  Call Extruder 0.17021
  MoveL (T15090) to (121.16, 113.18, 16.7) mm, rotated rx 180 ry 0 rz -180 deg; joints [1.945, 71.271, -37.578, 3.503, -33.743, -2.914]
  Call Extruder 0.01769
  MoveL (T15091) to (121.16, 113.76, 16.7) mm, rotated rx 180 ry 0 rz -180 deg; joints [1.945, 71.271, -37.578, 3.503, -33.743, -2.914]
  Call Extruder 0.17022
  MoveL (T15092) to (117.22, 109.83, 16.7) mm, rotated rx 180 ry 0 rz -180 deg; joints [3.284, 67.92, -31.274, 5.491, -36.773, -4.403]
  Call Extruder 0.01768
  MoveL (T15093) to (117.22, 110.41, 16.7) mm, rotated rx 180 ry 0 rz -180 deg; joints [3.284, 67.92, -31.274, 5.491, -36.773, -4.403]
  Call Extruder 0.17023
  MoveL (T15094) to (121.16, 114.34, 16.7) mm, rotated rx 180 ry 0 rz -180 deg; joints [3.287, 67.763, -30.978, 5.479, -36.911, -4.386]
  Call Extruder 0.01769
  MoveL (T15095) to (121.16, 114.92, 16.7) mm, rotated rx 180 ry 0 rz -180 deg; joints [3.287, 67.763, -30.978, 5.479, -36.911, -4.386]
  Call Extruder 0.11203
  MoveL (T15096) to (118.57, 112.33, 16.7) mm, rotated rx 180 ry 0 rz -180 deg; joints [1.884, 71.265, -37.567, 3.392, -33.745, -2.822]
  Call Extruder 0.01251
  MoveL (T15097) to (118.28, 112.62, 16.7) mm, rotated rx 180 ry 0 rz -180 deg; joints [1.823, 71.259, -37.556, 3.282, -33.747, -2.73]
  Call Extruder 0.12455
  MoveL (T15098) to (121.16, 115.5, 16.7) mm, rotated rx 180 ry 0 rz -180 deg; joints [1.823, 71.259, -37.556, 3.282, -33.747, -2.73]
  Call Extruder 0.01769
  MoveL (T15099) to (121.16, 116.08, 16.7) mm, rotated rx 180 ry 0 rz -180 deg; joints [3.291, 67.607, -30.685, 5.468, -37.048, -4.369]
  Call Extruder 0.13707
  MoveL (T15100) to (117.99, 112.91, 16.7) mm, rotated rx 180 ry 0 rz -180 deg; joints [3.295, 67.452, -30.393, 5.456, -37.184, -4.352]
  Call Extruder 0.01251
  MoveL (T15101) to (117.7, 113.2, 16.7) mm, rotated rx 180 ry 0 rz -180 deg; joints [3.295, 67.452, -30.393, 5.456, -37.184, -4.352]
  Call Extruder 0.1496
  MoveL (T15102) to (121.16, 116.65, 16.7) mm, rotated rx 180 ry 0 rz -180 deg; joints [3.295, 67.452, -30.393, 5.456, -37.184, -4.352]
  Call Extruder 0.01769
  MoveL (T15103) to (121.16, 117.23, 16.7) mm, rotated rx 180 ry 0 rz -180 deg; joints [1.762, 71.254, -37.545, 3.172, -33.75, -2.639]
  Call Extruder 0.16212
  MoveL (T15104) to (117.41, 113.48, 16.7) mm, rotated rx 180 ry 0 rz -180 deg; joints [1.762, 71.254, -37.545, 3.172, -33.75, -2.639]
  Call Extruder 0.00725
  MoveL (T15105) to (117.24, 113.65, 16.7) mm, rotated rx 180 ry 0 rz -180 deg; joints [1.701, 71.248, -37.534, 3.062, -33.752, -2.547]
  Call Extruder 0.00169
  MoveL (T15106) to (117.22, 113.7, 16.7) mm, rotated rx 180 ry 0 rz -180 deg; joints [1.701, 71.248, -37.534, 3.062, -33.752, -2.547]
  Call Extruder 0.00524
  MoveL (T15107) to (117.22, 113.88, 16.7) mm, rotated rx 180 ry 0 rz -180 deg; joints [3.298, 67.297, -30.102, 5.445, -37.32, -4.335]
  Call Extruder 0.17028
  MoveL (T15108) to (121.16, 117.81, 16.7) mm, rotated rx 180 ry 0 rz -180 deg; joints [3.298, 67.297, -30.102, 5.445, -37.32, -4.335]
  Call Extruder 0.01769
  MoveL (T15109) to (121.16, 118.39, 16.7) mm, rotated rx 180 ry 0 rz -180 deg; joints [3.302, 67.144, -29.813, 5.434, -37.455, -4.319]
  Call Extruder 0.1703
  MoveL (T15110) to (117.22, 114.45, 16.7) mm, rotated rx 180 ry 0 rz -180 deg; joints [3.302, 67.144, -29.813, 5.434, -37.455, -4.319]
  Call Extruder 0.01768
  MoveL (T15111) to (117.22, 115.03, 16.7) mm, rotated rx 180 ry 0 rz -180 deg; joints [3.302, 67.144, -29.813, 5.434, -37.455, -4.319]
  Call Extruder 0.17031
  MoveL (T15112) to (121.16, 118.97, 16.7) mm, rotated rx 180 ry 0 rz -180 deg; joints [1.64, 71.243, -37.525, 2.952, -33.754, -2.455]
  Call Extruder 0.01769
  MoveL (T15113) to (121.16, 119.55, 16.7) mm, rotated rx 180 ry 0 rz -180 deg; joints [1.64, 71.243, -37.525, 2.952, -33.754, -2.455]
  Call Extruder 0.17032
  MoveL (T15114) to (117.22, 115.61, 16.7) mm, rotated rx 180 ry 0 rz -180 deg; joints [1.64, 71.243, -37.525, 2.952, -33.754, -2.455]
  Call Extruder 0.01768
  MoveL (T15115) to (117.22, 116.19, 16.7) mm, rotated rx 180 ry 0 rz -180 deg; joints [1.579, 71.238, -37.515, 2.842, -33.756, -2.364]
  Call Extruder 0.17064
  MoveL (T15116) to (121.16, 120.14, 16.7) mm, rotated rx 180 ry 0 rz -180 deg; joints [1.579, 71.238, -37.515, 2.842, -33.756, -2.364]
  Call Extruder 0.01728
  MoveL (T15117) to (120.59, 120.14, 16.7) mm, rotated rx 180 ry 0 rz -180 deg; joints [3.305, 66.991, -29.526, 5.424, -37.589, -4.303]
  Call Extruder 0.14591
  MoveL (T15118) to (117.22, 116.76, 16.7) mm, rotated rx 180 ry 0 rz -180 deg; joints [3.305, 66.991, -29.526, 5.424, -37.589, -4.303]
  Call Extruder 0.01768
  MoveL (T15119) to (117.22, 117.34, 16.7) mm, rotated rx 180 ry 0 rz -180 deg; joints [3.309, 66.839, -29.241, 5.413, -37.722, -4.287]
  Call Extruder 0.12086
  MoveL (T15120) to (120.01, 120.14, 16.7) mm, rotated rx 180 ry 0 rz -180 deg; joints [3.309, 66.839, -29.241, 5.413, -37.722, -4.287]
  Call Extruder 0.01771
  MoveL (T15121) to (119.43, 120.14, 16.7) mm, rotated rx 180 ry 0 rz -180 deg; joints [3.309, 66.839, -29.241, 5.413, -37.722, -4.287]
  Call Extruder 0.10375
  MoveL (T15122) to (117.03, 117.74, 16.7) mm, rotated rx 180 ry 0 rz -180 deg; joints [3.309, 66.839, -29.241, 5.413, -37.722, -4.287]
  Set speed (45.0 mm/s)
  Call Extruder -1.6
  MoveL (T15123) to (117.03, 117.74, 16.7) mm, rotated rx 180 ry 0 rz -180 deg; joints [1.518, 71.233, -37.506, 2.732, -33.757, -2.272]
  Set speed (120.0 mm/s)
  MoveL (T15124) to (117.03, 117.74, 16.7) mm, rotated rx 180 ry 0 rz -180 deg; joints [1.518, 71.233, -37.506, 2.732, -33.757, -2.272]
  Call Extruder -0.38
  MoveL (T15125) to (117.79, 118.49, 16.7) mm, rotated rx 180 ry 0 rz -180 deg; joints [1.457, 71.228, -37.497, 2.622, -33.759, -2.181]
  Set speed (45.0 mm/s)
  Call Extruder -0.02
  MoveL (T15126) to (117.79, 118.49, 16.7) mm, rotated rx 180 ry 0 rz -180 deg; joints [1.457, 71.228, -37.497, 2.622, -33.759, -2.181]
  Set speed (150.0 mm/s)
  MoveL (T15127) to (117.79, 118.49, 18.7) mm, rotated rx 180 ry 0 rz -180 deg; joints [3.313, 66.688, -28.957, 5.403, -37.855, -4.271]
  MoveL (T15128) to (116.49, 107.94, 18.7) mm, rotated rx 180 ry 0 rz -180 deg; joints [3.313, 66.688, -28.957, 5.403, -37.855, -4.271]
  MoveL (T15129) to (116.49, 107.94, 16.7) mm, rotated rx 180 ry 0 rz -180 deg; joints [3.313, 66.688, -28.957, 5.403, -37.855, -4.271]
  Set speed (40.0 mm/s)
  Call Extruder 2.0
  MoveL (T15130) to (116.49, 107.94, 16.7) mm, rotated rx 180 ry 0 rz -180 deg; joints [3.313, 66.688, -28.957, 5.403, -37.855, -4.271]
  Set speed (37.7 mm/s)
  MoveL (T15131) to (116.49, 107.94, 16.7) mm, rotated rx 180 ry 0 rz -180 deg; joints [3.316, 66.538, -28.675, 5.393, -37.986, -4.255]
  Call Extruder 0.17708
  MoveL (T15132) to (112.39, 103.84, 16.7) mm, rotated rx 180 ry 0 rz -180 deg; joints [3.316, 66.538, -28.675, 5.393, -37.986, -4.255]
  Call Extruder 0.01769
  MoveL (T15133) to (111.82, 103.84, 16.7) mm, rotated rx 180 ry 0 rz -180 deg; joints [1.396, 71.223, -37.488, 2.512, -33.761, -2.089]
  Call Extruder 0.16915
  MoveL (T15134) to (115.72, 107.75, 16.7) mm, rotated rx 180 ry 0 rz -180 deg; joints [1.396, 71.223, -37.488, 2.512, -33.761, -2.089]
  Call Extruder 0.01769
  MoveL (T15135) to (115.15, 107.75, 16.7) mm, rotated rx 180 ry 0 rz -180 deg; joints [1.397, 71.043, -37.148, 2.505, -33.92, -2.079]
  Call Extruder 0.16915
  MoveL (T15136) to (111.24, 103.84, 16.7) mm, rotated rx 180 ry 0 rz -180 deg; joints [1.397, 71.043, -37.148, 2.505, -33.92, -2.079]
  Call Extruder 0.01769
  MoveL (T15137) to (110.66, 103.84, 16.7) mm, rotated rx 180 ry 0 rz -180 deg; joints [3.253, 66.53, -28.659, 5.29, -37.989, -4.174]
  Call Extruder 0.16915
  MoveL (T15138) to (114.57, 107.75, 16.7) mm, rotated rx 180 ry 0 rz -180 deg; joints [3.253, 66.53, -28.659, 5.29, -37.989, -4.174]
  Call Extruder 0.01769
  MoveL (T15139) to (113.99, 107.75, 16.7) mm, rotated rx 180 ry 0 rz -180 deg; joints [3.191, 66.521, -28.643, 5.188, -37.992, -4.093]
  Call Extruder 0.16915
  MoveL (T15140) to (110.08, 103.84, 16.7) mm, rotated rx 180 ry 0 rz -180 deg; joints [3.191, 66.521, -28.643, 5.188, -37.992, -4.093]
  Call Extruder 0.01769
  MoveL (T15141) to (109.5, 103.84, 16.7) mm, rotated rx 180 ry 0 rz -180 deg; joints [1.399, 70.864, -36.811, 2.497, -34.078, -2.069]
  Call Extruder 0.11483
  MoveL (T15142) to (112.16, 106.5, 16.7) mm, rotated rx 180 ry 0 rz -180 deg; joints [1.399, 70.864, -36.811, 2.497, -34.078, -2.069]
  Call Extruder 0.01251
  MoveL (T15143) to (111.87, 106.79, 16.7) mm, rotated rx 180 ry 0 rz -180 deg; joints [1.4, 70.686, -36.477, 2.49, -34.235, -2.059]
  Call Extruder 0.12733
  MoveL (T15144) to (108.92, 103.84, 16.7) mm, rotated rx 180 ry 0 rz -180 deg; joints [1.4, 70.686, -36.477, 2.49, -34.235, -2.059]
  Call Extruder 0.01769
  MoveL (T15145) to (108.35, 103.84, 16.7) mm, rotated rx 180 ry 0 rz -180 deg; joints [3.128, 66.513, -28.627, 5.085, -37.995, -4.011]
  Call Extruder 0.13984
  MoveL (T15146) to (111.58, 107.08, 16.7) mm, rotated rx 180 ry 0 rz -180 deg; joints [3.128, 66.513, -28.627, 5.085, -37.995, -4.011]
  Call Extruder 0.01251
  MoveL (T15147) to (111.29, 107.36, 16.7) mm, rotated rx 180 ry 0 rz -180 deg; joints [3.065, 66.505, -28.612, 4.982, -37.998, -3.93]
  Call Extruder 0.15235
  MoveL (T15148) to (107.77, 103.84, 16.7) mm, rotated rx 180 ry 0 rz -180 deg; joints [3.065, 66.505, -28.612, 4.982, -37.998, -3.93]
  Call Extruder 0.01769
  MoveL (T15149) to (107.19, 103.84, 16.7) mm, rotated rx 180 ry 0 rz -180 deg; joints [1.402, 70.51, -36.145, 2.483, -34.39, -2.049]
  Call Extruder 0.16485
  MoveL (T15150) to (111, 107.65, 16.7) mm, rotated rx 180 ry 0 rz -180 deg; joints [1.402, 70.51, -36.145, 2.483, -34.39, -2.049]
  Call Extruder 0.00339
  MoveL (T15151) to (110.92, 107.73, 16.7) mm, rotated rx 180 ry 0 rz -180 deg; joints [1.402, 70.51, -36.145, 2.483, -34.39, -2.049]
  Call Extruder 0.00168
  MoveL (T15152) to (110.87, 107.75, 16.7) mm, rotated rx 180 ry 0 rz -180 deg; joints [1.403, 70.335, -35.816, 2.476, -34.544, -2.039]
  Call Extruder 0.0107
  MoveL (T15153) to (110.52, 107.75, 16.7) mm, rotated rx 180 ry 0 rz -180 deg; joints [1.403, 70.335, -35.816, 2.476, -34.544, -2.039]
  Call Extruder 0.16915
  MoveL (T15154) to (106.61, 103.84, 16.7) mm, rotated rx 180 ry 0 rz -180 deg; joints [1.403, 70.335, -35.816, 2.476, -34.544, -2.039]
  Call Extruder 0.01769
  MoveL (T15155) to (106.03, 103.84, 16.7) mm, rotated rx 180 ry 0 rz -180 deg; joints [3.002, 66.497, -28.597, 4.88, -38, -3.849]
  Call Extruder 0.16915
  MoveL (T15156) to (109.94, 107.75, 16.7) mm, rotated rx 180 ry 0 rz -180 deg; joints [3.002, 66.497, -28.597, 4.88, -38, -3.849]
  Call Extruder 0.01769
  MoveL (T15157) to (109.36, 107.75, 16.7) mm, rotated rx 180 ry 0 rz -180 deg; joints [3.002, 66.497, -28.597, 4.88, -38, -3.849]
  Call Extruder 0.16915
  MoveL (T15158) to (105.45, 103.84, 16.7) mm, rotated rx 180 ry 0 rz -180 deg; joints [3.002, 66.497, -28.597, 4.88, -38, -3.849]
  Call Extruder 0.01769
  MoveL (T15159) to (104.88, 103.84, 16.7) mm, rotated rx 180 ry 0 rz -180 deg; joints [2.939, 66.489, -28.583, 4.777, -38.003, -3.768]
  Call Extruder 0.16915
  MoveL (T15160) to (108.79, 107.75, 16.7) mm, rotated rx 180 ry 0 rz -180 deg; joints [2.939, 66.489, -28.583, 4.777, -38.003, -3.768]
  Call Extruder 0.01769
  MoveL (T15161) to (108.21, 107.75, 16.7) mm, rotated rx 180 ry 0 rz -180 deg; joints [2.939, 66.489, -28.583, 4.777, -38.003, -3.768]
  Call Extruder 0.16005
  MoveL (T15162) to (104.51, 104.06, 16.7) mm, rotated rx 180 ry 0 rz -180 deg; joints [1.405, 70.161, -35.489, 2.469, -34.697, -2.03]
  Call Extruder 0.01768
  MoveL (T15163) to (104.51, 104.63, 16.7) mm, rotated rx 180 ry 0 rz -180 deg; joints [1.405, 70.161, -35.489, 2.469, -34.697, -2.03]
  Call Extruder 0.13504
  MoveL (T15164) to (107.63, 107.75, 16.7) mm, rotated rx 180 ry 0 rz -180 deg; joints [1.406, 69.989, -35.164, 2.462, -34.849, -2.021]
  Call Extruder 0.01769
  MoveL (T15165) to (107.05, 107.75, 16.7) mm, rotated rx 180 ry 0 rz -180 deg; joints [1.406, 69.989, -35.164, 2.462, -34.849, -2.021]
  Call Extruder 0.11004
  MoveL (T15166) to (104.51, 105.21, 16.7) mm, rotated rx 180 ry 0 rz -180 deg; joints [2.876, 66.482, -28.569, 4.675, -38.006, -3.686]
  Call Extruder 0.01678
  MoveL (T15167) to (104.51, 105.76, 16.7) mm, rotated rx 180 ry 0 rz -180 deg; joints [2.876, 66.482, -28.569, 4.675, -38.006, -3.686]
  Call Extruder 0.00167
  MoveL (T15168) to (104.53, 105.81, 16.7) mm, rotated rx 180 ry 0 rz -180 deg; joints [2.876, 66.482, -28.569, 4.675, -38.006, -3.686]
  Call Extruder 0.09205
  MoveL (T15169) to (106.66, 107.94, 16.7) mm, rotated rx 180 ry 0 rz -180 deg; joints [2.813, 66.474, -28.555, 4.572, -38.008, -3.605]
  Set speed (45.0 mm/s)
  Call Extruder -1.6
  MoveL (T15170) to (106.66, 107.94, 16.7) mm, rotated rx 180 ry 0 rz -180 deg; joints [2.813, 66.474, -28.555, 4.572, -38.008, -3.605]
  Set speed (120.0 mm/s)
  MoveL (T15171) to (106.66, 107.94, 16.7) mm, rotated rx 180 ry 0 rz -180 deg; joints [1.408, 69.817, -34.842, 2.455, -35, -2.012]
  Call Extruder -0.38
  MoveL (T15172) to (105.9, 107.18, 16.7) mm, rotated rx 180 ry 0 rz -180 deg; joints [1.408, 69.817, -34.842, 2.455, -35, -2.012]
  Set speed (45.0 mm/s)
  Call Extruder -0.02
  MoveL (T15173) to (105.9, 107.18, 16.7) mm, rotated rx 180 ry 0 rz -180 deg; joints [1.408, 69.817, -34.842, 2.455, -35, -2.012]
  Set speed (150.0 mm/s)
  MoveL (T15174) to (105.9, 107.18, 18.7) mm, rotated rx 180 ry 0 rz -180 deg; joints [1.409, 69.647, -34.523, 2.449, -35.149, -2.003]
  MoveL (T15175) to (104.34, 103.54, 18.7) mm, rotated rx 180 ry 0 rz -180 deg; joints [1.409, 69.647, -34.523, 2.449, -35.149, -2.003]
  MoveL (T15176) to (104.34, 103.54, 16.9) mm, rotated rx 180 ry 0 rz -180 deg; joints [2.751, 66.467, -28.541, 4.47, -38.011, -3.524]
  Set speed (40.0 mm/s)
  Call Extruder 2.0
  MoveL (T15177) to (104.34, 103.54, 16.9) mm, rotated rx 180 ry 0 rz -180 deg; joints [2.751, 66.467, -28.541, 4.47, -38.011, -3.524]
  Call Extruder 0.52159
  MoveL (T15178) to (121.46, 103.54, 16.9) mm, rotated rx 180 ry 0 rz -180 deg; joints [2.751, 66.467, -28.541, 4.47, -38.011, -3.524]
  Call Extruder 0.54596
  MoveL (T15179) to (121.46, 121.46, 16.9) mm, rotated rx 180 ry 0 rz -180 deg; joints [2.751, 66.467, -28.541, 4.47, -38.011, -3.524]
  Call Extruder 0.54596
  MoveL (T15180) to (103.54, 121.46, 16.9) mm, rotated rx 180 ry 0 rz -180 deg; joints [2.688, 66.46, -28.528, 4.367, -38.013, -3.443]
  Call Extruder 0.54596
  MoveL (T15181) to (103.54, 103.54, 16.9) mm, rotated rx 180 ry 0 rz -180 deg; joints [2.688, 66.46, -28.528, 4.367, -38.013, -3.443]
  Call Extruder 0.02254
  MoveL (T15182) to (104.28, 103.54, 16.9) mm, rotated rx 180 ry 0 rz -180 deg; joints [1.411, 69.479, -34.205, 2.442, -35.298, -1.994]
  Set speed (150.0 mm/s)
  MoveL (T15183) to (103.53, 103.13, 16.9) mm, rotated rx 180 ry 0 rz -180 deg; joints [1.411, 69.479, -34.205, 2.442, -35.298, -1.994]
  Set speed (40.0 mm/s)
  MoveL (T15184) to (103.53, 103.13, 16.9) mm, rotated rx 180 ry 0 rz -180 deg; joints [1.412, 69.311, -33.89, 2.436, -35.445, -1.985]
  Call Extruder 0.55858
  MoveL (T15185) to (121.87, 103.13, 16.9) mm, rotated rx 180 ry 0 rz -180 deg; joints [1.412, 69.311, -33.89, 2.436, -35.445, -1.985]
  Call Extruder 0.57077
  MoveL (T15186) to (121.87, 121.87, 16.9) mm, rotated rx 180 ry 0 rz -180 deg; joints [1.412, 69.311, -33.89, 2.436, -35.445, -1.985]
  Call Extruder 0.57077
  MoveL (T15187) to (103.13, 121.87, 16.9) mm, rotated rx 180 ry 0 rz -180 deg; joints [1.412, 69.311, -33.89, 2.436, -35.445, -1.985]
  Call Extruder 0.57077
  MoveL (T15188) to (103.13, 103.13, 16.9) mm, rotated rx 180 ry 0 rz -180 deg; joints [2.625, 66.453, -28.515, 4.264, -38.015, -3.362]
  Call Extruder 0.01036
  MoveL (T15189) to (103.47, 103.13, 16.9) mm, rotated rx 180 ry 0 rz -180 deg; joints [2.625, 66.453, -28.515, 4.264, -38.015, -3.362]
  Set speed (150.0 mm/s)
  MoveL (T15190) to (102.72, 102.81, 16.9) mm, rotated rx 180 ry 0 rz -180 deg; joints [2.562, 66.446, -28.502, 4.162, -38.018, -3.281]
  Set speed (25.0 mm/s)
  MoveL (T15191) to (102.72, 102.81, 16.9) mm, rotated rx 180 ry 0 rz -180 deg; joints [2.562, 66.446, -28.502, 4.162, -38.018, -3.281]
  Call Extruder 0.00259
  MoveL (T15192) to (102.72, 102.72, 16.9) mm, rotated rx 180 ry 0 rz -180 deg; joints [1.414, 69.145, -33.577, 2.43, -35.592, -1.976]
  Call Extruder 0.59557
  MoveL (T15193) to (122.28, 102.72, 16.9) mm, rotated rx 180 ry 0 rz -180 deg; joints [1.414, 69.145, -33.577, 2.43, -35.592, -1.976]
  Call Extruder 0.59557
  MoveL (T15194) to (122.28, 122.28, 16.9) mm, rotated rx 180 ry 0 rz -180 deg; joints [1.416, 68.98, -33.267, 2.424, -35.737, -1.968]
  Call Extruder 0.59557
  MoveL (T15195) to (102.72, 122.28, 16.9) mm, rotated rx 180 ry 0 rz -180 deg; joints [1.416, 68.98, -33.267, 2.424, -35.737, -1.968]
  Call Extruder 0.59115
  MoveL (T15196) to (102.72, 102.87, 16.9) mm, rotated rx 180 ry 0 rz -180 deg; joints [1.416, 68.98, -33.267, 2.424, -35.737, -1.968]
  Set speed (150.0 mm/s)
  MoveL (T15197) to (102.78, 102.75, 16.9) mm, rotated rx 180 ry 0 rz -180 deg; joints [2.499, 66.439, -28.489, 4.059, -38.02, -3.2]
  Set speed (45.0 mm/s)
  Call Extruder -1.6
  MoveL (T15198) to (102.78, 102.75, 16.9) mm, rotated rx 180 ry 0 rz -180 deg; joints [2.499, 66.439, -28.489, 4.059, -38.02, -3.2]
  Set speed (120.0 mm/s)
  MoveL (T15199) to (102.78, 102.75, 16.9) mm, rotated rx 180 ry 0 rz -180 deg; joints [2.436, 66.433, -28.477, 3.957, -38.022, -3.119]
  Call Extruder -0.05166
  MoveL (T15200) to (102.72, 102.72, 16.9) mm, rotated rx 180 ry 0 rz -180 deg; joints [2.436, 66.433, -28.477, 3.957, -38.022, -3.119]
  Call Extruder -0.32834
  MoveL (T15201) to (103.65, 102.72, 16.9) mm, rotated rx 180 ry 0 rz -180 deg; joints [1.417, 68.816, -32.958, 2.418, -35.882, -1.96]
  Set speed (45.0 mm/s)
  Call Extruder -0.02
  MoveL (T15202) to (103.65, 102.72, 16.9) mm, rotated rx 180 ry 0 rz -180 deg; joints [1.419, 68.653, -32.652, 2.412, -36.025, -1.952]
  Set speed (150.0 mm/s)
  MoveL (T15203) to (103.65, 102.72, 18.9) mm, rotated rx 180 ry 0 rz -180 deg; joints [1.419, 68.653, -32.652, 2.412, -36.025, -1.952]
  MoveL (T15204) to (103.84, 106.29, 18.9) mm, rotated rx 180 ry 0 rz -180 deg; joints [2.373, 66.427, -28.466, 3.855, -38.024, -3.038]
  MoveL (T15205) to (103.84, 106.29, 16.9) mm, rotated rx 180 ry 0 rz -180 deg; joints [2.373, 66.427, -28.466, 3.855, -38.024, -3.038]
  Set speed (40.0 mm/s)
  Call Extruder 2.0
  MoveL (T15206) to (103.84, 106.29, 16.9) mm, rotated rx 180 ry 0 rz -180 deg; joints [2.373, 66.427, -28.466, 3.855, -38.024, -3.038]
  Set speed (50.0 mm/s)
  MoveL (T15207) to (103.84, 106.29, 16.9) mm, rotated rx 180 ry 0 rz -180 deg; joints [2.31, 66.421, -28.454, 3.752, -38.026, -2.957]
  Call Extruder 0.07441
  MoveL (T15208) to (103.84, 103.84, 16.9) mm, rotated rx 180 ry 0 rz -180 deg; joints [2.31, 66.421, -28.454, 3.752, -38.026, -2.957]
  Call Extruder 0.0111
  MoveL (T15209) to (104.1, 104.1, 16.9) mm, rotated rx 180 ry 0 rz -180 deg; joints [2.31, 66.421, -28.454, 3.752, -38.026, -2.957]
  Call Extruder 0.05294
  MoveL (T15210) to (104.1, 105.84, 16.9) mm, rotated rx 180 ry 0 rz -180 deg; joints [1.42, 68.491, -32.347, 2.407, -36.168, -1.943]
  Call Extruder 0.00661
  MoveL (T15211) to (104.18, 106.04, 16.9) mm, rotated rx 180 ry 0 rz -180 deg; joints [1.42, 68.491, -32.347, 2.407, -36.168, -1.943]
  Call Extruder 0.02065
  MoveL (T15212) to (104.66, 106.52, 16.9) mm, rotated rx 180 ry 0 rz -180 deg; joints [1.42, 68.491, -32.347, 2.407, -36.168, -1.943]
  Call Extruder 0.03528
  MoveL (T15213) to (103.84, 107.34, 16.9) mm, rotated rx 180 ry 0 rz -180 deg; joints [1.422, 68.33, -32.044, 2.401, -36.31, -1.935]
  Call Extruder 0.03385
  MoveL (T15214) to (103.84, 108.45, 16.9) mm, rotated rx 180 ry 0 rz -180 deg; joints [1.422, 68.33, -32.044, 2.401, -36.31, -1.935]
  Call Extruder 0.13495
  MoveL (T15215) to (106.98, 111.58, 16.9) mm, rotated rx 180 ry 0 rz -180 deg; joints [1.422, 68.33, -32.044, 2.401, -36.31, -1.935]
  Call Extruder 0.04156
  MoveL (T15216) to (107.6, 112.8, 16.9) mm, rotated rx 180 ry 0 rz -180 deg; joints [1.422, 68.33, -32.044, 2.401, -36.31, -1.935]
  Call Extruder 0.16166
  MoveL (T15217) to (103.84, 116.55, 16.9) mm, rotated rx 180 ry 0 rz -180 deg; joints [2.247, 66.415, -28.443, 3.65, -38.028, -2.876]
  Call Extruder 0.03385
  MoveL (T15218) to (103.84, 117.66, 16.9) mm, rotated rx 180 ry 0 rz -180 deg; joints [2.247, 66.415, -28.443, 3.65, -38.028, -2.876]
  Call Extruder 0.05612
  MoveL (T15219) to (105.15, 118.96, 16.9) mm, rotated rx 180 ry 0 rz -180 deg; joints [2.185, 66.409, -28.432, 3.547, -38.03, -2.796]
  Call Extruder 0.02709
  MoveL (T15220) to (105.15, 119.85, 16.9) mm, rotated rx 180 ry 0 rz -180 deg; joints [2.185, 66.409, -28.432, 3.547, -38.03, -2.796]
  Call Extruder 0.05612
  MoveL (T15221) to (103.84, 121.16, 16.9) mm, rotated rx 180 ry 0 rz -180 deg; joints [2.185, 66.409, -28.432, 3.547, -38.03, -2.796]
  Call Extruder 0.06345
  MoveL (T15222) to (105.93, 121.16, 16.9) mm, rotated rx 180 ry 0 rz -180 deg; joints [1.423, 68.17, -31.744, 2.396, -36.45, -1.928]
  Call Extruder 0.01096
  MoveL (T15223) to (105.67, 120.9, 16.9) mm, rotated rx 180 ry 0 rz -180 deg; joints [1.423, 68.17, -31.744, 2.396, -36.45, -1.928]
  Set speed (45.0 mm/s)
  Call Extruder -1.6
  MoveL (T15224) to (105.67, 120.9, 16.9) mm, rotated rx 180 ry 0 rz -180 deg; joints [1.425, 68.011, -31.445, 2.391, -36.59, -1.92]
  Set speed (120.0 mm/s)
  MoveL (T15225) to (105.67, 120.9, 16.9) mm, rotated rx 180 ry 0 rz -180 deg; joints [1.425, 68.011, -31.445, 2.391, -36.59, -1.92]
  Call Extruder -0.12811
  MoveL (T15226) to (105.93, 121.16, 16.9) mm, rotated rx 180 ry 0 rz -180 deg; joints [2.122, 66.403, -28.422, 3.445, -38.032, -2.715]
  Call Extruder -0.25189
  MoveL (T15227) to (105.22, 121.16, 16.9) mm, rotated rx 180 ry 0 rz -180 deg; joints [2.122, 66.403, -28.422, 3.445, -38.032, -2.715]
  Set speed (45.0 mm/s)
  Call Extruder -0.02
  MoveL (T15228) to (105.22, 121.16, 16.9) mm, rotated rx 180 ry 0 rz -180 deg; joints [2.122, 66.403, -28.422, 3.445, -38.032, -2.715]
  Set speed (150.0 mm/s)
  MoveL (T15229) to (105.22, 121.16, 18.9) mm, rotated rx 180 ry 0 rz -180 deg; joints [2.059, 66.398, -28.411, 3.342, -38.034, -2.634]
  MoveL (T15230) to (105.15, 117.23, 18.9) mm, rotated rx 180 ry 0 rz -180 deg; joints [2.059, 66.398, -28.411, 3.342, -38.034, -2.634]
  MoveL (T15231) to (105.15, 117.23, 16.9) mm, rotated rx 180 ry 0 rz -180 deg; joints [2.059, 66.398, -28.411, 3.342, -38.034, -2.634]
  Set speed (40.0 mm/s)
  Call Extruder 2.0
  MoveL (T15232) to (105.15, 117.23, 16.9) mm, rotated rx 180 ry 0 rz -180 deg; joints [1.426, 67.853, -31.148, 2.385, -36.729, -1.912]
  Set speed (50.0 mm/s)
  MoveL (T15233) to (105.15, 117.23, 16.9) mm, rotated rx 180 ry 0 rz -180 deg; joints [1.426, 67.853, -31.148, 2.385, -36.729, -1.912]
  Call Extruder 0.04143
  MoveL (T15234) to (105.15, 115.87, 16.9) mm, rotated rx 180 ry 0 rz -180 deg; joints [1.426, 67.853, -31.148, 2.385, -36.729, -1.912]
  Call Extruder 0.00661
  MoveL (T15235) to (105.23, 115.67, 16.9) mm, rotated rx 180 ry 0 rz -180 deg; joints [1.428, 67.696, -30.852, 2.38, -36.867, -1.905]
  Call Extruder 0.02637
  MoveL (T15236) to (105.84, 115.05, 16.9) mm, rotated rx 180 ry 0 rz -180 deg; joints [1.428, 67.696, -30.852, 2.38, -36.867, -1.905]
  Call Extruder 0.08606
  MoveL (T15237) to (103.84, 113.06, 16.9) mm, rotated rx 180 ry 0 rz -180 deg; joints [1.428, 67.696, -30.852, 2.38, -36.867, -1.905]
  Call Extruder 0.03385
  MoveL (T15238) to (103.84, 111.94, 16.9) mm, rotated rx 180 ry 0 rz -180 deg; joints [1.428, 67.696, -30.852, 2.38, -36.867, -1.905]
  Call Extruder 0.09463
  MoveL (T15239) to (106.04, 109.75, 16.9) mm, rotated rx 180 ry 0 rz -180 deg; joints [1.996, 66.393, -28.401, 3.24, -38.036, -2.553]
  Call Extruder 0.05062
  MoveL (T15240) to (105.29, 108.27, 16.9) mm, rotated rx 180 ry 0 rz -180 deg; joints [1.996, 66.393, -28.401, 3.24, -38.036, -2.553]
  Call Extruder 0.02377
  MoveL (T15241) to (105.1, 107.51, 16.9) mm, rotated rx 180 ry 0 rz -180 deg; joints [1.996, 66.393, -28.401, 3.24, -38.036, -2.553]
  Set speed (45.0 mm/s)
  Call Extruder -1.6
  MoveL (T15242) to (105.1, 107.51, 16.9) mm, rotated rx 180 ry 0 rz -180 deg; joints [1.933, 66.388, -28.392, 3.138, -38.037, -2.472]
  Set speed (120.0 mm/s)
  MoveL (T15243) to (105.1, 107.51, 16.9) mm, rotated rx 180 ry 0 rz -180 deg; joints [1.933, 66.388, -28.392, 3.138, -38.037, -2.472]
  Call Extruder -0.27797
  MoveL (T15244) to (105.29, 108.27, 16.9) mm, rotated rx 180 ry 0 rz -180 deg; joints [1.429, 67.54, -30.559, 2.375, -37.005, -1.897]
  Call Extruder -0.10203
  MoveL (T15245) to (105.42, 108.52, 16.9) mm, rotated rx 180 ry 0 rz -180 deg; joints [1.429, 67.54, -30.559, 2.375, -37.005, -1.897]
  Set speed (45.0 mm/s)
  Call Extruder -0.02
  MoveL (T15246) to (105.42, 108.52, 16.9) mm, rotated rx 180 ry 0 rz -180 deg; joints [1.429, 67.54, -30.559, 2.375, -37.005, -1.897]
  Set speed (150.0 mm/s)
  MoveL (T15247) to (105.42, 108.52, 18.9) mm, rotated rx 180 ry 0 rz -180 deg; joints [1.429, 67.54, -30.559, 2.375, -37.005, -1.897]
  MoveL (T15248) to (117.45, 112.15, 18.9) mm, rotated rx 180 ry 0 rz -180 deg; joints [1.431, 67.385, -30.267, 2.37, -37.141, -1.89]
  MoveL (T15249) to (117.45, 112.15, 16.9) mm, rotated rx 180 ry 0 rz -180 deg; joints [1.431, 67.385, -30.267, 2.37, -37.141, -1.89]
  Set speed (40.0 mm/s)
  Call Extruder 2.0
  MoveL (T15250) to (117.45, 112.15, 16.9) mm, rotated rx 180 ry 0 rz -180 deg; joints [1.87, 66.383, -28.382, 3.035, -38.039, -2.391]
  Set speed (50.0 mm/s)
  MoveL (T15251) to (117.45, 112.15, 16.9) mm, rotated rx 180 ry 0 rz -180 deg; joints [1.807, 66.378, -28.373, 2.933, -38.041, -2.311]
  Call Extruder 0.01607
  MoveL (T15252) to (117.83, 111.78, 16.9) mm, rotated rx 180 ry 0 rz -180 deg; joints [1.807, 66.378, -28.373, 2.933, -38.041, -2.311]
  Set speed (45.0 mm/s)
  Call Extruder -1.6
  MoveL (T15253) to (117.83, 111.78, 16.9) mm, rotated rx 180 ry 0 rz -180 deg; joints [1.807, 66.378, -28.373, 2.933, -38.041, -2.311]
  Set speed (120.0 mm/s)
  MoveL (T15254) to (117.83, 111.78, 16.9) mm, rotated rx 180 ry 0 rz -180 deg; joints [1.807, 66.378, -28.373, 2.933, -38.041, -2.311]
  Call Extruder -0.18789
  MoveL (T15255) to (117.45, 112.15, 16.9) mm, rotated rx 180 ry 0 rz -180 deg; joints [1.433, 67.231, -29.977, 2.366, -37.277, -1.883]
  Set speed (45.0 mm/s)
  Call Extruder -0.21211
  MoveL (T15256) to (117.45, 112.15, 16.9) mm, rotated rx 180 ry 0 rz -180 deg; joints [1.433, 67.231, -29.977, 2.366, -37.277, -1.883]
  Set speed (150.0 mm/s)
  MoveL (T15257) to (117.45, 112.15, 18.9) mm, rotated rx 180 ry 0 rz -180 deg; joints [1.434, 67.077, -29.689, 2.361, -37.412, -1.876]
  MoveL (T15258) to (121.34, 119.42, 18.9) mm, rotated rx 180 ry 0 rz -180 deg; joints [1.434, 67.077, -29.689, 2.361, -37.412, -1.876]
  MoveL (T15259) to (121.34, 119.42, 16.9) mm, rotated rx 180 ry 0 rz -180 deg; joints [1.744, 66.373, -28.365, 2.831, -38.042, -2.23]
  Set speed (40.0 mm/s)
  Call Extruder 2.0
  MoveL (T15260) to (121.34, 119.42, 16.9) mm, rotated rx 180 ry 0 rz -180 deg; joints [1.744, 66.373, -28.365, 2.831, -38.042, -2.23]
  Call Extruder 0.03108
  MoveL (T15261) to (120.62, 120.14, 16.9) mm, rotated rx 180 ry 0 rz -180 deg; joints [1.744, 66.373, -28.365, 2.831, -38.042, -2.23]
  Call Extruder 0.01774
  MoveL (T15262) to (120.04, 120.14, 16.9) mm, rotated rx 180 ry 0 rz -180 deg; joints [1.681, 66.369, -28.356, 2.728, -38.044, -2.149]
  Call Extruder 0.04823
  MoveL (T15263) to (121.16, 119.02, 16.9) mm, rotated rx 180 ry 0 rz -180 deg; joints [1.681, 66.369, -28.356, 2.728, -38.044, -2.149]
  Call Extruder 0.01777
  MoveL (T15264) to (121.16, 118.44, 16.9) mm, rotated rx 180 ry 0 rz -180 deg; joints [1.436, 66.925, -29.402, 2.356, -37.546, -1.869]
  Call Extruder 0.07952
  MoveL (T15265) to (119.32, 120.28, 16.9) mm, rotated rx 180 ry 0 rz -180 deg; joints [1.436, 66.925, -29.402, 2.356, -37.546, -1.869]
  Call Extruder 0.01256
  MoveL (T15266) to (119.03, 119.99, 16.9) mm, rotated rx 180 ry 0 rz -180 deg; joints [1.437, 66.773, -29.117, 2.352, -37.679, -1.862]
  Call Extruder 0.09207
  MoveL (T15267) to (121.16, 117.86, 16.9) mm, rotated rx 180 ry 0 rz -180 deg; joints [1.437, 66.773, -29.117, 2.352, -37.679, -1.862]
  Call Extruder 0.01777
  MoveL (T15268) to (121.16, 117.28, 16.9) mm, rotated rx 180 ry 0 rz -180 deg; joints [1.437, 66.773, -29.117, 2.352, -37.679, -1.862]
  Call Extruder 0.10462
  MoveL (T15269) to (118.74, 119.7, 16.9) mm, rotated rx 180 ry 0 rz -180 deg; joints [1.437, 66.773, -29.117, 2.352, -37.679, -1.862]
  Call Extruder 0.01256
  MoveL (T15270) to (118.45, 119.41, 16.9) mm, rotated rx 180 ry 0 rz -180 deg; joints [1.618, 66.364, -28.348, 2.626, -38.045, -2.069]
  Call Extruder 0.11718
  MoveL (T15271) to (121.16, 116.7, 16.9) mm, rotated rx 180 ry 0 rz -180 deg; joints [1.555, 66.36, -28.341, 2.524, -38.047, -1.988]
  Call Extruder 0.01777
  MoveL (T15272) to (121.16, 116.13, 16.9) mm, rotated rx 180 ry 0 rz -180 deg; joints [1.555, 66.36, -28.341, 2.524, -38.047, -1.988]
  Call Extruder 0.12973
  MoveL (T15273) to (118.16, 119.12, 16.9) mm, rotated rx 180 ry 0 rz -180 deg; joints [1.555, 66.36, -28.341, 2.524, -38.047, -1.988]
  Call Extruder 0.01256
  MoveL (T15274) to (117.87, 118.83, 16.9) mm, rotated rx 180 ry 0 rz -180 deg; joints [1.439, 66.623, -28.834, 2.347, -37.812, -1.855]
  Call Extruder 0.14228
  MoveL (T15275) to (121.16, 115.55, 16.9) mm, rotated rx 180 ry 0 rz -180 deg; joints [1.439, 66.623, -28.834, 2.347, -37.812, -1.855]
  Call Extruder 0.01777
  MoveL (T15276) to (121.16, 114.97, 16.9) mm, rotated rx 180 ry 0 rz -180 deg; joints [1.44, 66.473, -28.552, 2.343, -37.944, -1.848]
  Call Extruder 0.15483
  MoveL (T15277) to (117.58, 118.54, 16.9) mm, rotated rx 180 ry 0 rz -180 deg; joints [1.44, 66.473, -28.552, 2.343, -37.944, -1.848]
  Call Extruder 0.01256
  MoveL (T15278) to (117.3, 118.25, 16.9) mm, rotated rx 180 ry 0 rz -180 deg; joints [1.512, 66.311, -28.247, 2.452, -38.089, -1.931]
  Call Extruder 0.16739
  MoveL (T15279) to (121.16, 114.39, 16.9) mm, rotated rx 180 ry 0 rz -180 deg; joints [1.512, 66.311, -28.247, 2.452, -38.089, -1.931]
  Call Extruder 0.01777
  MoveL (T15280) to (121.16, 113.81, 16.9) mm, rotated rx 180 ry 0 rz -180 deg; joints [1.512, 66.311, -28.247, 2.452, -38.089, -1.931]
  Call Extruder 0.17073
  MoveL (T15281) to (117.22, 117.75, 16.9) mm, rotated rx 180 ry 0 rz -180 deg; joints [1.512, 66.311, -28.247, 2.452, -38.089, -1.931]
  Call Extruder 0.01778
  MoveL (T15282) to (117.22, 117.17, 16.9) mm, rotated rx 180 ry 0 rz -180 deg; joints [1.512, 66.311, -28.247, 2.452, -38.089, -1.931]
  Call Extruder 0.17072
  MoveL (T15283) to (121.16, 113.23, 16.9) mm, rotated rx 180 ry 0 rz -180 deg; joints [1.512, 66.311, -28.247, 2.452, -38.089, -1.931]
  Call Extruder 0.01777
  MoveL (T15284) to (121.16, 112.65, 16.9) mm, rotated rx 180 ry 0 rz -180 deg; joints [1.512, 66.311, -28.247, 2.452, -38.089, -1.931]
  Call Extruder 0.1707
  MoveL (T15285) to (117.22, 116.59, 16.9) mm, rotated rx 180 ry 0 rz -180 deg; joints [1.44, 66.473, -28.552, 2.343, -37.944, -1.848]
  Call Extruder 0.01778
  MoveL (T15286) to (117.22, 116.01, 16.9) mm, rotated rx 180 ry 0 rz -180 deg; joints [1.44, 66.473, -28.552, 2.343, -37.944, -1.848]
  Call Extruder 0.17069
  MoveL (T15287) to (121.16, 112.07, 16.9) mm, rotated rx 180 ry 0 rz -180 deg; joints [1.44, 66.512, -28.625, 2.344, -37.91, -1.85]
  Call Extruder 0.01777
  MoveL (T15288) to (121.16, 111.49, 16.9) mm, rotated rx 180 ry 0 rz -180 deg; joints [1.44, 66.512, -28.625, 2.344, -37.91, -1.85]
  Call Extruder 0.17068
  MoveL (T15289) to (117.22, 115.43, 16.9) mm, rotated rx 180 ry 0 rz -180 deg; joints [1.44, 66.512, -28.625, 2.344, -37.91, -1.85]
  Call Extruder 0.01778
  MoveL (T15290) to (117.22, 114.85, 16.9) mm, rotated rx 180 ry 0 rz -180 deg; joints [1.44, 66.512, -28.625, 2.344, -37.91, -1.85]
  Call Extruder 0.17067
  MoveL (T15291) to (121.16, 110.91, 16.9) mm, rotated rx 180 ry 0 rz -180 deg; joints [1.44, 66.512, -28.625, 2.344, -37.91, -1.85]
  Call Extruder 0.01777
  MoveL (T15292) to (121.16, 110.33, 16.9) mm, rotated rx 180 ry 0 rz -180 deg; joints [1.44, 66.512, -28.625, 2.344, -37.91, -1.85]
  Call Extruder 0.17066
  MoveL (T15293) to (117.22, 114.27, 16.9) mm, rotated rx 180 ry 0 rz -180 deg; joints [1.44, 66.512, -28.625, 2.344, -37.91, -1.85]
  Call Extruder 0.01813
  MoveL (T15294) to (117.23, 113.68, 16.9) mm, rotated rx 180 ry 0 rz -180 deg; joints [1.44, 66.512, -28.625, 2.344, -37.91, -1.85]
  Call Extruder 0.17015
  MoveL (T15295) to (121.16, 109.75, 16.9) mm, rotated rx 180 ry 0 rz -180 deg; joints [1.407, 66.455, -28.559, 2.29, -37.918, -1.807]
  Call Extruder 0.01777
  MoveL (T15296) to (121.16, 109.17, 16.9) mm, rotated rx 180 ry 0 rz -180 deg; joints [1.407, 66.455, -28.559, 2.29, -37.918, -1.807]
  Call Extruder 0.11319
  MoveL (T15297) to (118.55, 111.78, 16.9) mm, rotated rx 180 ry 0 rz -180 deg; joints [1.407, 66.455, -28.559, 2.29, -37.918, -1.807]
  Call Extruder 0.01256
  MoveL (T15298) to (118.26, 111.49, 16.9) mm, rotated rx 180 ry 0 rz -180 deg; joints [1.407, 66.455, -28.559, 2.29, -37.918, -1.807]
  Call Extruder 0.12575
  MoveL (T15299) to (121.16, 108.59, 16.9) mm, rotated rx 180 ry 0 rz -180 deg; joints [1.407, 66.455, -28.559, 2.29, -37.918, -1.807]
  Call Extruder 0.01777
  MoveL (T15300) to (121.16, 108.01, 16.9) mm, rotated rx 180 ry 0 rz -180 deg; joints [1.363, 71.293, -37.659, 2.46, -33.659, -2.048]
  Call Extruder 0.14563
  MoveL (T15301) to (117.8, 111.37, 16.9) mm, rotated rx 180 ry 0 rz -180 deg; joints [1.363, 71.293, -37.659, 2.46, -33.659, -2.048]
  Call Extruder 0.01767
  MoveL (T15302) to (117.22, 111.37, 16.9) mm, rotated rx 180 ry 0 rz -180 deg; joints [3.241, 71.52, -38.086, 5.869, -33.573, -4.895]
  Call Extruder 0.17069
  MoveL (T15303) to (121.16, 107.43, 16.9) mm, rotated rx 180 ry 0 rz -180 deg; joints [3.241, 71.52, -38.086, 5.869, -33.573, -4.895]
  Call Extruder 0.01777
  MoveL (T15304) to (121.16, 106.86, 16.9) mm, rotated rx 180 ry 0 rz -180 deg; joints [3.351, 66.44, -28.532, 5.444, -38.034, -4.293]
  Call Extruder 0.17061
  MoveL (T15305) to (117.22, 110.79, 16.9) mm, rotated rx 180 ry 0 rz -180 deg; joints [3.351, 66.44, -28.532, 5.444, -38.034, -4.293]
  Call Extruder 0.01778
  MoveL (T15306) to (117.22, 110.21, 16.9) mm, rotated rx 180 ry 0 rz -180 deg; joints [3.351, 66.44, -28.532, 5.444, -38.034, -4.293]
  Call Extruder 0.1706
  MoveL (T15307) to (121.16, 106.28, 16.9) mm, rotated rx 180 ry 0 rz -180 deg; joints [3.351, 66.44, -28.532, 5.444, -38.034, -4.293]
  Call Extruder 0.01777
  MoveL (T15308) to (121.16, 105.7, 16.9) mm, rotated rx 180 ry 0 rz -180 deg; joints [1.409, 66.249, -28.173, 2.285, -38.099, -1.798]
  Call Extruder 0.17058
  MoveL (T15309) to (117.22, 109.63, 16.9) mm, rotated rx 180 ry 0 rz -180 deg; joints [1.409, 66.249, -28.173, 2.285, -38.099, -1.798]
  Call Extruder 0.01778
  MoveL (T15310) to (117.22, 109.05, 16.9) mm, rotated rx 180 ry 0 rz -180 deg; joints [1.409, 66.249, -28.173, 2.285, -38.099, -1.798]
  Call Extruder 0.17057
  MoveL (T15311) to (121.16, 105.12, 16.9) mm, rotated rx 180 ry 0 rz -180 deg; joints [1.407, 66.439, -28.53, 2.29, -37.932, -1.807]
  Call Extruder 0.01777
  MoveL (T15312) to (121.16, 104.54, 16.9) mm, rotated rx 180 ry 0 rz -180 deg; joints [1.407, 66.439, -28.53, 2.29, -37.932, -1.807]
  Call Extruder 0.17056
  MoveL (T15313) to (117.22, 108.47, 16.9) mm, rotated rx 180 ry 0 rz -180 deg; joints [1.407, 66.439, -28.53, 2.29, -37.932, -1.807]
  Call Extruder 0.01778
  MoveL (T15314) to (117.22, 107.89, 16.9) mm, rotated rx 180 ry 0 rz -180 deg; joints [1.365, 66.245, -28.165, 2.213, -38.101, -1.742]
  Call Extruder 0.16962
  MoveL (T15315) to (121.13, 103.98, 16.9) mm, rotated rx 180 ry 0 rz -180 deg; joints [1.365, 66.245, -28.165, 2.213, -38.101, -1.742]
  Call Extruder 0.01778
  MoveL (T15316) to (120.55, 103.98, 16.9) mm, rotated rx 180 ry 0 rz -180 deg; joints [1.365, 66.245, -28.165, 2.213, -38.101, -1.742]
  Call Extruder 0.16368
  MoveL (T15317) to (116.78, 107.75, 16.9) mm, rotated rx 180 ry 0 rz -180 deg; joints [1.365, 66.245, -28.165, 2.213, -38.101, -1.742]
  Call Extruder 0.01777
  MoveL (T15318) to (116.2, 107.75, 16.9) mm, rotated rx 180 ry 0 rz -180 deg; joints [1.365, 66.245, -28.165, 2.213, -38.101, -1.742]
  Call Extruder 0.16367
  MoveL (T15319) to (119.97, 103.98, 16.9) mm, rotated rx 180 ry 0 rz -180 deg; joints [1.319, 71.418, -37.894, 2.388, -33.547, -1.991]
  Call Extruder 0.00371
  MoveL (T15320) to (119.85, 103.98, 16.9) mm, rotated rx 180 ry 0 rz -180 deg; joints [1.319, 71.418, -37.894, 2.388, -33.547, -1.991]
  Call Extruder 0.00414
  MoveL (T15321) to (119.85, 103.84, 16.9) mm, rotated rx 180 ry 0 rz -180 deg; joints [1.319, 71.418, -37.894, 2.388, -33.547, -1.991]
  Call Extruder 0.00992
  MoveL (T15322) to (119.53, 103.84, 16.9) mm, rotated rx 180 ry 0 rz -180 deg; joints [3.282, 71.657, -38.343, 5.96, -33.457, -4.978]
  Call Extruder 0.16951
  MoveL (T15323) to (115.62, 107.75, 16.9) mm, rotated rx 180 ry 0 rz -180 deg; joints [3.398, 66.342, -28.347, 5.509, -38.124, -4.339]
  Call Extruder 0.01777
  MoveL (T15324) to (115.04, 107.75, 16.9) mm, rotated rx 180 ry 0 rz -180 deg; joints [3.398, 66.342, -28.347, 5.509, -38.124, -4.339]
  Call Extruder 0.16951
  MoveL (T15325) to (118.95, 103.84, 16.9) mm, rotated rx 180 ry 0 rz -180 deg; joints [3.398, 66.342, -28.347, 5.509, -38.124, -4.339]
  Call Extruder 0.01777
  MoveL (T15326) to (118.37, 103.84, 16.9) mm, rotated rx 180 ry 0 rz -180 deg; joints [1.366, 66.143, -27.973, 2.21, -38.191, -1.737]
  Call Extruder 0.16951
  MoveL (T15327) to (114.46, 107.75, 16.9) mm, rotated rx 180 ry 0 rz -180 deg; joints [1.366, 66.143, -27.973, 2.21, -38.191, -1.737]
  Call Extruder 0.01777
  MoveL (T15328) to (113.88, 107.75, 16.9) mm, rotated rx 180 ry 0 rz -180 deg; joints [1.365, 66.23, -28.136, 2.213, -38.115, -1.741]
  Call Extruder 0.16951
  MoveL (T15329) to (117.79, 103.84, 16.9) mm, rotated rx 180 ry 0 rz -180 deg; joints [1.365, 66.23, -28.136, 2.213, -38.115, -1.741]
  Call Extruder 0.01777
  MoveL (T15330) to (117.21, 103.84, 16.9) mm, rotated rx 180 ry 0 rz -180 deg; joints [1.332, 66.038, -27.775, 2.151, -38.282, -1.689]
  Call Extruder 0.16599
  MoveL (T15331) to (113.38, 107.67, 16.9) mm, rotated rx 180 ry 0 rz -180 deg; joints [1.332, 66.038, -27.775, 2.151, -38.282, -1.689]
  Call Extruder 0.01256
  MoveL (T15332) to (113.09, 107.38, 16.9) mm, rotated rx 180 ry 0 rz -180 deg; joints [1.332, 66.038, -27.775, 2.151, -38.282, -1.689]
  Call Extruder 0.15343
  MoveL (T15333) to (116.63, 103.84, 16.9) mm, rotated rx 180 ry 0 rz -180 deg; joints [1.332, 66.038, -27.775, 2.151, -38.282, -1.689]
  Call Extruder 0.01777
  MoveL (T15334) to (116.05, 103.84, 16.9) mm, rotated rx 180 ry 0 rz -180 deg; joints [1.332, 66.038, -27.775, 2.151, -38.282, -1.689]
  Call Extruder 0.14087
  MoveL (T15335) to (112.81, 107.09, 16.9) mm, rotated rx 180 ry 0 rz -180 deg; joints [1.332, 66.038, -27.775, 2.151, -38.282, -1.689]
  Call Extruder 0.01256
  MoveL (T15336) to (112.52, 106.8, 16.9) mm, rotated rx 180 ry 0 rz -180 deg; joints [1.323, 66.037, -27.774, 2.136, -38.283, -1.677]
  Call Extruder 0.12831
  MoveL (T15337) to (115.47, 103.84, 16.9) mm, rotated rx 180 ry 0 rz -180 deg; joints [1.323, 66.037, -27.774, 2.136, -38.283, -1.677]
  Call Extruder 0.01777
  MoveL (T15338) to (114.89, 103.84, 16.9) mm, rotated rx 180 ry 0 rz -180 deg; joints [1.276, 71.544, -38.131, 2.316, -33.435, -1.933]
  Call Extruder 0.11574
  MoveL (T15339) to (112.22, 106.51, 16.9) mm, rotated rx 180 ry 0 rz -180 deg; joints [1.276, 71.544, -38.131, 2.316, -33.435, -1.933]
  Call Extruder 0.00182
  MoveL (T15340) to (112.18, 106.47, 16.9) mm, rotated rx 180 ry 0 rz -180 deg; joints [3.322, 71.795, -38.602, 6.051, -33.34, -5.061]
  Call Extruder 0.05469
  MoveL (T15341) to (110.92, 107.73, 16.9) mm, rotated rx 180 ry 0 rz -180 deg; joints [3.322, 71.795, -38.602, 6.051, -33.34, -5.061]
  Call Extruder 0.00169
  MoveL (T15342) to (110.87, 107.75, 16.9) mm, rotated rx 180 ry 0 rz -180 deg; joints [3.322, 71.795, -38.602, 6.051, -33.34, -5.061]
  Call Extruder 0.01426
  MoveL (T15343) to (110.41, 107.75, 16.9) mm, rotated rx 180 ry 0 rz -180 deg; joints [3.445, 66.244, -28.163, 5.574, -38.213, -4.385]
  Call Extruder 0.16951
  MoveL (T15344) to (114.31, 103.84, 16.9) mm, rotated rx 180 ry 0 rz -180 deg; joints [3.445, 66.244, -28.163, 5.574, -38.213, -4.385]
  Call Extruder 0.01777
  MoveL (T15345) to (113.73, 103.84, 16.9) mm, rotated rx 180 ry 0 rz -180 deg; joints [1.339, 66.038, -27.776, 2.162, -38.282, -1.697]
  Call Extruder 0.16951
  MoveL (T15346) to (109.83, 107.75, 16.9) mm, rotated rx 180 ry 0 rz -180 deg; joints [1.339, 66.038, -27.776, 2.162, -38.282, -1.697]
  Call Extruder 0.01777
  MoveL (T15347) to (109.25, 107.75, 16.9) mm, rotated rx 180 ry 0 rz -180 deg; joints [1.339, 66.038, -27.776, 2.162, -38.282, -1.697]
  Call Extruder 0.16951
  MoveL (T15348) to (113.16, 103.84, 16.9) mm, rotated rx 180 ry 0 rz -180 deg; joints [1.326, 66.053, -27.803, 2.141, -38.269, -1.681]
  Call Extruder 0.01777
  MoveL (T15349) to (112.58, 103.84, 16.9) mm, rotated rx 180 ry 0 rz -180 deg; joints [1.326, 66.053, -27.803, 2.141, -38.269, -1.681]
  Call Extruder 0.16951
  MoveL (T15350) to (108.67, 107.75, 16.9) mm, rotated rx 180 ry 0 rz -180 deg; joints [1.326, 66.053, -27.803, 2.141, -38.269, -1.681]
  Call Extruder 0.01777
  MoveL (T15351) to (108.09, 107.75, 16.9) mm, rotated rx 180 ry 0 rz -180 deg; joints [1.326, 66.053, -27.803, 2.141, -38.269, -1.681]
  Call Extruder 0.16951
  MoveL (T15352) to (112, 103.84, 16.9) mm, rotated rx 180 ry 0 rz -180 deg; joints [1.326, 66.053, -27.803, 2.141, -38.269, -1.681]
  Call Extruder 0.01777
  MoveL (T15353) to (111.42, 103.84, 16.9) mm, rotated rx 180 ry 0 rz -180 deg; joints [1.326, 66.053, -27.803, 2.141, -38.269, -1.681]
  Call Extruder 0.16951
  MoveL (T15354) to (107.51, 107.75, 16.9) mm, rotated rx 180 ry 0 rz -180 deg; joints [1.326, 66.053, -27.803, 2.141, -38.269, -1.681]
  Call Extruder 0.01777
  MoveL (T15355) to (106.93, 107.75, 16.9) mm, rotated rx 180 ry 0 rz -180 deg; joints [1.326, 66.053, -27.803, 2.141, -38.269, -1.681]
  Call Extruder 0.16951
  MoveL (T15356) to (110.84, 103.84, 16.9) mm, rotated rx 180 ry 0 rz -180 deg; joints [1.326, 66.053, -27.803, 2.141, -38.269, -1.681]
  Call Extruder 0.01777
  MoveL (T15357) to (110.26, 103.84, 16.9) mm, rotated rx 180 ry 0 rz -180 deg; joints [1.326, 66.053, -27.803, 2.141, -38.269, -1.681]
  Call Extruder 0.16951
  MoveL (T15358) to (106.35, 107.75, 16.9) mm, rotated rx 180 ry 0 rz -180 deg; joints [1.323, 66.037, -27.774, 2.136, -38.283, -1.677]
  Call Extruder 0.01777
  MoveL (T15359) to (105.77, 107.75, 16.9) mm, rotated rx 180 ry 0 rz -180 deg; joints [1.321, 66.272, -28.216, 2.142, -38.076, -1.687]
  Call Extruder 0.16951
  MoveL (T15360) to (109.68, 103.84, 16.9) mm, rotated rx 180 ry 0 rz -180 deg; joints [1.321, 66.272, -28.216, 2.142, -38.076, -1.687]
  Call Extruder 0.01777
  MoveL (T15361) to (109.1, 103.84, 16.9) mm, rotated rx 180 ry 0 rz -180 deg; joints [1.321, 66.272, -28.216, 2.142, -38.076, -1.687]
  Call Extruder 0.15614
  MoveL (T15362) to (105.5, 107.44, 16.9) mm, rotated rx 180 ry 0 rz -180 deg; joints [1.321, 66.272, -28.216, 2.142, -38.076, -1.687]
  Call Extruder 0.00405
  MoveL (T15363) to (105.47, 107.32, 16.9) mm, rotated rx 180 ry 0 rz -180 deg; joints [1.321, 66.272, -28.216, 2.142, -38.076, -1.687]
  Call Extruder 0.01293
  MoveL (T15364) to (105.47, 106.89, 16.9) mm, rotated rx 180 ry 0 rz -180 deg; joints [1.321, 66.272, -28.216, 2.142, -38.076, -1.687]
  Call Extruder 0.13227
  MoveL (T15365) to (108.52, 103.84, 16.9) mm, rotated rx 180 ry 0 rz -180 deg; joints [1.321, 66.272, -28.216, 2.142, -38.076, -1.687]
  Call Extruder 0.01777
  MoveL (T15366) to (107.94, 103.84, 16.9) mm, rotated rx 180 ry 0 rz -180 deg; joints [1.321, 66.034, -28.177, 2.152, -37.877, -1.699]
  Call Extruder 0.11659
  MoveL (T15367) to (105.25, 106.53, 16.9) mm, rotated rx 180 ry 0 rz -180 deg; joints [1.378, 70.763, -37.056, 2.483, -33.731, -2.065]
  Call Extruder 0.01256
  MoveL (T15368) to (104.96, 106.24, 16.9) mm, rotated rx 180 ry 0 rz -180 deg; joints [1.378, 70.997, -37.102, 2.471, -33.92, -2.051]
  Call Extruder 0.10402
  MoveL (T15369) to (107.36, 103.84, 16.9) mm, rotated rx 180 ry 0 rz -180 deg; joints [1.378, 70.997, -37.102, 2.471, -33.92, -2.051]
  Call Extruder 0.01777
  MoveL (T15370) to (106.78, 103.84, 16.9) mm, rotated rx 180 ry 0 rz -180 deg; joints [1.378, 70.997, -37.102, 2.471, -33.92, -2.051]
  Call Extruder 0.09145
  MoveL (T15371) to (104.67, 105.95, 16.9) mm, rotated rx 180 ry 0 rz -180 deg; joints [1.378, 70.997, -37.102, 2.471, -33.92, -2.051]
  Call Extruder 0.00622
  MoveL (T15372) to (104.53, 105.81, 16.9) mm, rotated rx 180 ry 0 rz -180 deg; joints [1.445, 71.204, -37.49, 2.602, -33.741, -2.164]
  Call Extruder 0.00169
  MoveL (T15373) to (104.51, 105.76, 16.9) mm, rotated rx 180 ry 0 rz -180 deg; joints [1.445, 71.204, -37.49, 2.602, -33.741, -2.164]
  Call Extruder 0.00677
  MoveL (T15374) to (104.51, 105.54, 16.9) mm, rotated rx 180 ry 0 rz -180 deg; joints [1.506, 71.208, -37.499, 2.712, -33.739, -2.256]
  Call Extruder 0.07345
  MoveL (T15375) to (106.2, 103.84, 16.9) mm, rotated rx 180 ry 0 rz -180 deg; joints [1.506, 71.208, -37.499, 2.712, -33.739, -2.256]
  Call Extruder 0.01777
  MoveL (T15376) to (105.62, 103.84, 16.9) mm, rotated rx 180 ry 0 rz -180 deg; joints [1.399, 70.876, -36.874, 2.5, -34.028, -2.072]
  Call Extruder 0.04831
  MoveL (T15377) to (104.51, 104.96, 16.9) mm, rotated rx 180 ry 0 rz -180 deg; joints [1.399, 70.876, -36.874, 2.5, -34.028, -2.072]
  Call Extruder 0.01778
  MoveL (T15378) to (104.51, 104.38, 16.9) mm, rotated rx 180 ry 0 rz -180 deg; joints [1.4, 70.698, -36.539, 2.492, -34.185, -2.062]
  Call Extruder 0.03112
  MoveL (T15379) to (105.23, 103.66, 16.9) mm, rotated rx 180 ry 0 rz -180 deg; joints [1.4, 70.698, -36.539, 2.492, -34.185, -2.062]
  Set speed (45.0 mm/s)
  Call Extruder -1.6
  MoveL (T15380) to (105.23, 103.66, 16.9) mm, rotated rx 180 ry 0 rz -180 deg; joints [1.4, 70.698, -36.539, 2.492, -34.185, -2.062]
  Set speed (120.0 mm/s)
  MoveL (T15381) to (105.23, 103.66, 16.9) mm, rotated rx 180 ry 0 rz -180 deg; joints [1.567, 71.213, -37.508, 2.822, -33.737, -2.347]
  Call Extruder -0.36151
  MoveL (T15382) to (104.51, 104.38, 16.9) mm, rotated rx 180 ry 0 rz -180 deg; joints [1.567, 71.213, -37.508, 2.822, -33.737, -2.347]
  Call Extruder -0.01849
  MoveL (T15383) to (104.51, 104.43, 16.9) mm, rotated rx 180 ry 0 rz -180 deg; joints [1.628, 71.218, -37.518, 2.932, -33.735, -2.439]
  Set speed (45.0 mm/s)
  Call Extruder -0.02
  MoveL (T15384) to (104.51, 104.43, 16.9) mm, rotated rx 180 ry 0 rz -180 deg; joints [1.628, 71.218, -37.518, 2.932, -33.735, -2.439]
  Set speed (150.0 mm/s)
  MoveL (T15385) to (104.51, 104.43, 18.9) mm, rotated rx 180 ry 0 rz -180 deg; joints [1.402, 70.521, -36.206, 2.485, -34.34, -2.052]
  MoveL (T15386) to (119.38, 120.65, 18.9) mm, rotated rx 180 ry 0 rz -180 deg; joints [1.402, 70.521, -36.206, 2.485, -34.34, -2.052]
  MoveL (T15387) to (119.38, 120.65, 16.9) mm, rotated rx 180 ry 0 rz -180 deg; joints [1.402, 70.521, -36.206, 2.485, -34.34, -2.052]
  Set speed (40.0 mm/s)
  Call Extruder 2.0
  MoveL (T15388) to (119.38, 120.65, 16.9) mm, rotated rx 180 ry 0 rz -180 deg; joints [1.403, 70.346, -35.876, 2.478, -34.494, -2.043]
  Set speed (25.0 mm/s)
  MoveL (T15389) to (119.38, 120.65, 16.9) mm, rotated rx 180 ry 0 rz -180 deg; joints [1.403, 70.346, -35.876, 2.478, -34.494, -2.043]
  Call Extruder 0.02011
  MoveL (T15390) to (118.84, 121.19, 16.9) mm, rotated rx 180 ry 0 rz -180 deg; joints [1.689, 71.224, -37.528, 3.042, -33.733, -2.53]
  Call Extruder 0.01314
  MoveL (T15391) to (118.34, 121.19, 16.9) mm, rotated rx 180 ry 0 rz -180 deg; joints [1.689, 71.224, -37.528, 3.042, -33.733, -2.53]
  Call Extruder 0.02531
  MoveL (T15392) to (119.02, 120.51, 16.9) mm, rotated rx 180 ry 0 rz -180 deg; joints [1.689, 71.224, -37.528, 3.042, -33.733, -2.53]
  Call Extruder 0.00929
  MoveL (T15393) to (118.77, 120.26, 16.9) mm, rotated rx 180 ry 0 rz -180 deg; joints [1.75, 71.229, -37.538, 3.152, -33.731, -2.622]
  Call Extruder 0.0346
  MoveL (T15394) to (117.84, 121.19, 16.9) mm, rotated rx 180 ry 0 rz -180 deg; joints [1.75, 71.229, -37.538, 3.152, -33.731, -2.622]
  Call Extruder 0.01314
  MoveL (T15395) to (117.34, 121.19, 16.9) mm, rotated rx 180 ry 0 rz -180 deg; joints [1.405, 70.172, -35.55, 2.471, -34.647, -2.033]
  Call Extruder 0.0439
  MoveL (T15396) to (118.52, 120.01, 16.9) mm, rotated rx 180 ry 0 rz -180 deg; joints [1.405, 70.172, -35.55, 2.471, -34.647, -2.033]
  Call Extruder 0.00929
  MoveL (T15397) to (118.27, 119.76, 16.9) mm, rotated rx 180 ry 0 rz -180 deg; joints [1.406, 70, -35.225, 2.464, -34.799, -2.024]
  Call Extruder 0.05319
  MoveL (T15398) to (116.85, 121.19, 16.9) mm, rotated rx 180 ry 0 rz -180 deg; joints [1.406, 70, -35.225, 2.464, -34.799, -2.024]
  Call Extruder 0.01314
  MoveL (T15399) to (116.35, 121.19, 16.9) mm, rotated rx 180 ry 0 rz -180 deg; joints [1.811, 71.235, -37.548, 3.262, -33.729, -2.714]
  Call Extruder 0.06249
  MoveL (T15400) to (118.02, 119.51, 16.9) mm, rotated rx 180 ry 0 rz -180 deg; joints [1.811, 71.235, -37.548, 3.262, -33.729, -2.714]
  Call Extruder 0.00929
  MoveL (T15401) to (117.78, 119.26, 16.9) mm, rotated rx 180 ry 0 rz -180 deg; joints [1.811, 71.235, -37.548, 3.262, -33.729, -2.714]
  Call Extruder 0.07179
  MoveL (T15402) to (115.85, 121.19, 16.9) mm, rotated rx 180 ry 0 rz -180 deg; joints [1.811, 71.235, -37.548, 3.262, -33.729, -2.714]
  Call Extruder 0.01314
  MoveL (T15403) to (115.35, 121.19, 16.9) mm, rotated rx 180 ry 0 rz -180 deg; joints [1.871, 71.241, -37.559, 3.372, -33.727, -2.805]
  Call Extruder 0.08108
  MoveL (T15404) to (117.53, 119.01, 16.9) mm, rotated rx 180 ry 0 rz -180 deg; joints [1.408, 69.828, -34.903, 2.458, -34.95, -2.015]
  Call Extruder 0.00929
  MoveL (T15405) to (117.28, 118.76, 16.9) mm, rotated rx 180 ry 0 rz -180 deg; joints [1.408, 69.828, -34.903, 2.458, -34.95, -2.015]
  Call Extruder 0.09038
  MoveL (T15406) to (114.85, 121.19, 16.9) mm, rotated rx 180 ry 0 rz -180 deg; joints [1.409, 69.658, -34.582, 2.451, -35.1, -2.006]
  Call Extruder 0.01314
  MoveL (T15407) to (114.36, 121.19, 16.9) mm, rotated rx 180 ry 0 rz -180 deg; joints [1.409, 69.658, -34.582, 2.451, -35.1, -2.006]
  Call Extruder 0.09967
  MoveL (T15408) to (117.03, 118.51, 16.9) mm, rotated rx 180 ry 0 rz -180 deg; joints [1.932, 71.247, -37.571, 3.482, -33.725, -2.897]
  Call Extruder 0.00403
  MoveL (T15409) to (116.92, 118.4, 16.9) mm, rotated rx 180 ry 0 rz -180 deg; joints [1.932, 71.247, -37.571, 3.482, -33.725, -2.897]
  Call Extruder 0.00575
  MoveL (T15410) to (116.84, 118.2, 16.9) mm, rotated rx 180 ry 0 rz -180 deg; joints [1.932, 71.247, -37.571, 3.482, -33.725, -2.897]
  Call Extruder 0.11131
  MoveL (T15411) to (113.86, 121.19, 16.9) mm, rotated rx 180 ry 0 rz -180 deg; joints [1.993, 71.253, -37.583, 3.592, -33.722, -2.989]
  Call Extruder 0.01314
  MoveL (T15412) to (113.36, 121.19, 16.9) mm, rotated rx 180 ry 0 rz -180 deg; joints [1.993, 71.253, -37.583, 3.592, -33.722, -2.989]
  Call Extruder 0.12989
  MoveL (T15413) to (116.84, 117.7, 16.9) mm, rotated rx 180 ry 0 rz -180 deg; joints [1.411, 69.489, -34.265, 2.445, -35.249, -1.997]
  Call Extruder 0.01314
  MoveL (T15414) to (116.84, 117.2, 16.9) mm, rotated rx 180 ry 0 rz -180 deg; joints [1.411, 69.489, -34.265, 2.445, -35.249, -1.997]
  Call Extruder 0.14847
  MoveL (T15415) to (112.86, 121.19, 16.9) mm, rotated rx 180 ry 0 rz -180 deg; joints [1.412, 69.321, -33.949, 2.439, -35.397, -1.988]
  Call Extruder 0.01314
  MoveL (T15416) to (112.36, 121.19, 16.9) mm, rotated rx 180 ry 0 rz -180 deg; joints [2.054, 71.259, -37.595, 3.702, -33.72, -3.081]
  Call Extruder 0.16706
  MoveL (T15417) to (116.84, 116.7, 16.9) mm, rotated rx 180 ry 0 rz -180 deg; joints [2.054, 71.259, -37.595, 3.702, -33.72, -3.081]
  Call Extruder 0.01314
  MoveL (T15418) to (116.84, 116.21, 16.9) mm, rotated rx 180 ry 0 rz -180 deg; joints [2.115, 71.266, -37.607, 3.813, -33.717, -3.173]
  Call Extruder 0.18564
  MoveL (T15419) to (111.86, 121.19, 16.9) mm, rotated rx 180 ry 0 rz -180 deg; joints [2.115, 71.266, -37.607, 3.813, -33.717, -3.173]
  Call Extruder 0.01314
  MoveL (T15420) to (111.36, 121.19, 16.9) mm, rotated rx 180 ry 0 rz -180 deg; joints [1.414, 69.155, -33.636, 2.432, -35.543, -1.98]
  Call Extruder 0.20423
  MoveL (T15421) to (116.84, 115.71, 16.9) mm, rotated rx 180 ry 0 rz -180 deg; joints [1.414, 69.155, -33.636, 2.432, -35.543, -1.98]
  Call Extruder 0.01314
  MoveL (T15422) to (116.84, 115.21, 16.9) mm, rotated rx 180 ry 0 rz -180 deg; joints [1.415, 68.989, -33.325, 2.426, -35.689, -1.971]
  Call Extruder 0.22281
  MoveL (T15423) to (110.87, 121.19, 16.9) mm, rotated rx 180 ry 0 rz -180 deg; joints [1.415, 68.989, -33.325, 2.426, -35.689, -1.971]
  Call Extruder 0.01314
  MoveL (T15424) to (110.37, 121.19, 16.9) mm, rotated rx 180 ry 0 rz -180 deg; joints [2.176, 71.273, -37.62, 3.923, -33.715, -3.265]
  Call Extruder 0.2414
  MoveL (T15425) to (116.84, 114.71, 16.9) mm, rotated rx 180 ry 0 rz -180 deg; joints [2.237, 71.28, -37.633, 4.033, -33.712, -3.357]
  Call Extruder 0.01314
  MoveL (T15426) to (116.84, 114.21, 16.9) mm, rotated rx 180 ry 0 rz -180 deg; joints [2.237, 71.28, -37.633, 4.033, -33.712, -3.357]
  Call Extruder 0.25998
  MoveL (T15427) to (109.87, 121.19, 16.9) mm, rotated rx 180 ry 0 rz -180 deg; joints [2.237, 71.28, -37.633, 4.033, -33.712, -3.357]
  Call Extruder 0.01314
  MoveL (T15428) to (109.37, 121.19, 16.9) mm, rotated rx 180 ry 0 rz -180 deg; joints [1.417, 68.825, -33.015, 2.421, -35.834, -1.963]
  Call Extruder 0.27856
  MoveL (T15429) to (116.84, 113.72, 16.9) mm, rotated rx 180 ry 0 rz -180 deg; joints [1.417, 68.825, -33.015, 2.421, -35.834, -1.963]
  Call Extruder 0.00228
  MoveL (T15430) to (116.84, 113.63, 16.9) mm, rotated rx 180 ry 0 rz -180 deg; joints [1.417, 68.825, -33.015, 2.421, -35.834, -1.963]
  Call Extruder 0.0054
  MoveL (T15431) to (116.92, 113.44, 16.9) mm, rotated rx 180 ry 0 rz -180 deg; joints [1.418, 68.662, -32.708, 2.415, -35.977, -1.955]
  Call Extruder 0.01891
  MoveL (T15432) to (117.43, 112.93, 16.9) mm, rotated rx 180 ry 0 rz -180 deg; joints [1.418, 68.662, -32.708, 2.415, -35.977, -1.955]
  Call Extruder 0.00591
  MoveL (T15433) to (117.33, 112.73, 16.9) mm, rotated rx 180 ry 0 rz -180 deg; joints [2.298, 71.287, -37.647, 4.143, -33.709, -3.449]
  Call Extruder 0.31519
  MoveL (T15434) to (108.87, 121.19, 16.9) mm, rotated rx 180 ry 0 rz -180 deg; joints [2.298, 71.287, -37.647, 4.143, -33.709, -3.449]
  Call Extruder 0.01314
  MoveL (T15435) to (108.38, 121.19, 16.9) mm, rotated rx 180 ry 0 rz -180 deg; joints [2.359, 71.294, -37.661, 4.254, -33.707, -3.541]
  Call Extruder 0.32748
  MoveL (T15436) to (117.16, 112.4, 16.9) mm, rotated rx 180 ry 0 rz -180 deg; joints [2.359, 71.294, -37.661, 4.254, -33.707, -3.541]
  Call Extruder 0.00976
  MoveL (T15437) to (116.99, 112.07, 16.9) mm, rotated rx 180 ry 0 rz -180 deg; joints [1.42, 68.499, -32.403, 2.409, -36.12, -1.946]
  Call Extruder 0.33977
  MoveL (T15438) to (107.88, 121.19, 16.9) mm, rotated rx 180 ry 0 rz -180 deg; joints [1.42, 68.499, -32.403, 2.409, -36.12, -1.946]
  Call Extruder 0.01314
  MoveL (T15439) to (107.38, 121.19, 16.9) mm, rotated rx 180 ry 0 rz -180 deg; joints [1.421, 68.338, -32.1, 2.404, -36.262, -1.938]
  Call Extruder 0.35637
  MoveL (T15440) to (116.94, 111.63, 16.9) mm, rotated rx 180 ry 0 rz -180 deg; joints [1.421, 68.338, -32.1, 2.404, -36.262, -1.938]
  Set speed (150.0 mm/s)
  MoveL (T15441) to (117, 111.07, 16.9) mm, rotated rx 180 ry 0 rz -180 deg; joints [1.421, 68.338, -32.1, 2.404, -36.262, -1.938]
  Set speed (25.0 mm/s)
  MoveL (T15442) to (117, 111.07, 16.9) mm, rotated rx 180 ry 0 rz -180 deg; joints [2.42, 71.302, -37.675, 4.364, -33.704, -3.633]
  Call Extruder 0.37728
  MoveL (T15443) to (106.88, 121.19, 16.9) mm, rotated rx 180 ry 0 rz -180 deg; joints [2.42, 71.302, -37.675, 4.364, -33.704, -3.633]
  Call Extruder 0.01031
  MoveL (T15444) to (106.49, 121.19, 16.9) mm, rotated rx 180 ry 0 rz -180 deg; joints [2.481, 71.31, -37.69, 4.474, -33.701, -3.725]
  Call Extruder 0.002
  MoveL (T15445) to (106.44, 121.13, 16.9) mm, rotated rx 180 ry 0 rz -180 deg; joints [2.481, 71.31, -37.69, 4.474, -33.701, -3.725]
  Call Extruder 0.38806
  MoveL (T15446) to (116.84, 110.72, 16.9) mm, rotated rx 180 ry 0 rz -180 deg; joints [2.481, 71.31, -37.69, 4.474, -33.701, -3.725]
  Call Extruder 0.01314
  MoveL (T15447) to (116.84, 110.23, 16.9) mm, rotated rx 180 ry 0 rz -180 deg; joints [1.423, 68.178, -31.799, 2.398, -36.403, -1.931]
  Call Extruder 0.39735
  MoveL (T15448) to (106.19, 120.88, 16.9) mm, rotated rx 180 ry 0 rz -180 deg; joints [1.423, 68.178, -31.799, 2.398, -36.403, -1.931]
  Call Extruder 0.00929
  MoveL (T15449) to (105.94, 120.63, 16.9) mm, rotated rx 180 ry 0 rz -180 deg; joints [1.424, 68.019, -31.5, 2.393, -36.543, -1.923]
  Call Extruder 0.40665
  MoveL (T15450) to (116.84, 109.73, 16.9) mm, rotated rx 180 ry 0 rz -180 deg; joints [1.424, 68.019, -31.5, 2.393, -36.543, -1.923]
  Call Extruder 0.01314
  MoveL (T15451) to (116.84, 109.23, 16.9) mm, rotated rx 180 ry 0 rz -180 deg; joints [1.424, 68.019, -31.5, 2.393, -36.543, -1.923]
  Call Extruder 0.41595
  MoveL (T15452) to (105.69, 120.39, 16.9) mm, rotated rx 180 ry 0 rz -180 deg; joints [2.542, 71.318, -37.705, 4.584, -33.698, -3.817]
  Call Extruder 0.00522
  MoveL (T15453) to (105.55, 120.25, 16.9) mm, rotated rx 180 ry 0 rz -180 deg; joints [2.542, 71.318, -37.705, 4.584, -33.698, -3.817]
  Call Extruder 0.00177
  MoveL (T15454) to (105.52, 120.18, 16.9) mm, rotated rx 180 ry 0 rz -180 deg; joints [2.603, 71.326, -37.72, 4.695, -33.695, -3.909]
  Call Extruder 0.00343
  MoveL (T15455) to (105.52, 120.05, 16.9) mm, rotated rx 180 ry 0 rz -180 deg; joints [2.603, 71.326, -37.72, 4.695, -33.695, -3.909]
  Call Extruder 0.42214
  MoveL (T15456) to (116.85, 108.73, 16.9) mm, rotated rx 180 ry 0 rz -180 deg; joints [2.603, 71.326, -37.72, 4.695, -33.695, -3.909]
  Call Extruder 0.01314
  MoveL (T15457) to (116.85, 108.23, 16.9) mm, rotated rx 180 ry 0 rz -180 deg; joints [1.426, 67.861, -31.203, 2.388, -36.682, -1.915]
  Call Extruder 0.42215
  MoveL (T15458) to (105.52, 119.55, 16.9) mm, rotated rx 180 ry 0 rz -180 deg; joints [1.426, 67.861, -31.203, 2.388, -36.682, -1.915]
  Call Extruder 0.01314
  MoveL (T15459) to (105.52, 119.06, 16.9) mm, rotated rx 180 ry 0 rz -180 deg; joints [1.426, 67.861, -31.203, 2.388, -36.682, -1.915]
  Call Extruder 0.40738
  MoveL (T15460) to (116.45, 108.13, 16.9) mm, rotated rx 180 ry 0 rz -180 deg; joints [1.428, 67.704, -30.907, 2.382, -36.82, -1.908]
  Call Extruder 0.01314
  MoveL (T15461) to (115.95, 108.13, 16.9) mm, rotated rx 180 ry 0 rz -180 deg; joints [1.428, 67.704, -30.907, 2.382, -36.82, -1.908]
  Call Extruder 0.3888
  MoveL (T15462) to (105.52, 118.56, 16.9) mm, rotated rx 180 ry 0 rz -180 deg; joints [1.428, 67.704, -30.907, 2.382, -36.82, -1.908]
  Call Extruder 0.01314
  MoveL (T15463) to (105.52, 118.06, 16.9) mm, rotated rx 180 ry 0 rz -180 deg; joints [2.663, 71.334, -37.736, 4.805, -33.692, -4.001]
  Call Extruder 0.37022
  MoveL (T15464) to (115.45, 108.13, 16.9) mm, rotated rx 180 ry 0 rz -180 deg; joints [2.663, 71.334, -37.736, 4.805, -33.692, -4.001]
  Call Extruder 0.01314
  MoveL (T15465) to (114.95, 108.13, 16.9) mm, rotated rx 180 ry 0 rz -180 deg; joints [2.663, 71.334, -37.736, 4.805, -33.692, -4.001]
  Call Extruder 0.35165
  MoveL (T15466) to (105.52, 117.56, 16.9) mm, rotated rx 180 ry 0 rz -180 deg; joints [2.724, 71.343, -37.752, 4.916, -33.688, -4.093]
  Call Extruder 0.01314
  MoveL (T15467) to (105.52, 117.06, 16.9) mm, rotated rx 180 ry 0 rz -180 deg; joints [2.724, 71.343, -37.752, 4.916, -33.688, -4.093]
  Call Extruder 0.33307
  MoveL (T15468) to (114.46, 108.13, 16.9) mm, rotated rx 180 ry 0 rz -180 deg; joints [1.429, 67.548, -30.614, 2.377, -36.958, -1.9]
  Call Extruder 0.01314
  MoveL (T15469) to (113.96, 108.13, 16.9) mm, rotated rx 180 ry 0 rz -180 deg; joints [1.429, 67.548, -30.614, 2.377, -36.958, -1.9]
  Call Extruder 0.20542
  MoveL (T15470) to (108.45, 113.64, 16.9) mm, rotated rx 180 ry 0 rz -180 deg; joints [1.429, 67.548, -30.614, 2.377, -36.958, -1.9]
  Call Extruder 0.00838
  MoveL (T15471) to (108.59, 113.92, 16.9) mm, rotated rx 180 ry 0 rz -180 deg; joints [1.431, 67.392, -30.321, 2.373, -37.094, -1.893]
  Call Extruder 0.01127
  MoveL (T15472) to (108.17, 113.92, 16.9) mm, rotated rx 180 ry 0 rz -180 deg; joints [1.431, 67.392, -30.321, 2.373, -37.094, -1.893]
  Call Extruder 0.09852
  MoveL (T15473) to (105.52, 116.56, 16.9) mm, rotated rx 180 ry 0 rz -180 deg; joints [2.785, 71.352, -37.768, 5.026, -33.685, -4.186]
  Call Extruder 0.01314
  MoveL (T15474) to (105.52, 116.07, 16.9) mm, rotated rx 180 ry 0 rz -180 deg; joints [2.785, 71.352, -37.768, 5.026, -33.685, -4.186]
  Call Extruder 0.08575
  MoveL (T15475) to (107.82, 113.77, 16.9) mm, rotated rx 180 ry 0 rz -180 deg; joints [2.785, 71.352, -37.768, 5.026, -33.685, -4.186]
  Set speed (150.0 mm/s)
  MoveL (T15476) to (108.17, 113.43, 16.9) mm, rotated rx 180 ry 0 rz -180 deg; joints [2.846, 71.361, -37.785, 5.137, -33.682, -4.278]
  Set speed (25.0 mm/s)
  MoveL (T15477) to (108.17, 113.43, 16.9) mm, rotated rx 180 ry 0 rz -180 deg; joints [2.846, 71.361, -37.785, 5.137, -33.682, -4.278]
  Call Extruder 0.19744
  MoveL (T15478) to (113.46, 108.13, 16.9) mm, rotated rx 180 ry 0 rz -180 deg; joints [2.846, 71.361, -37.785, 5.137, -33.682, -4.278]
  Call Extruder 0.00105
  MoveL (T15479) to (113.42, 108.13, 16.9) mm, rotated rx 180 ry 0 rz -180 deg; joints [2.846, 71.361, -37.785, 5.137, -33.682, -4.278]
  Call Extruder 0.0054
  MoveL (T15480) to (113.23, 108.05, 16.9) mm, rotated rx 180 ry 0 rz -180 deg; joints [1.432, 67.238, -30.031, 2.368, -37.23, -1.886]
  Call Extruder 0.00356
  MoveL (T15481) to (113.14, 107.96, 16.9) mm, rotated rx 180 ry 0 rz -180 deg; joints [1.432, 67.238, -30.031, 2.368, -37.23, -1.886]
  Call Extruder 0.1873
  MoveL (T15482) to (108.11, 112.98, 16.9) mm, rotated rx 180 ry 0 rz -180 deg; joints [1.434, 67.084, -29.742, 2.363, -37.365, -1.878]
  Call Extruder 0.00976
  MoveL (T15483) to (107.94, 112.65, 16.9) mm, rotated rx 180 ry 0 rz -180 deg; joints [1.434, 67.084, -29.742, 2.363, -37.365, -1.878]
  Call Extruder 0.18429
  MoveL (T15484) to (112.89, 107.71, 16.9) mm, rotated rx 180 ry 0 rz -180 deg; joints [2.907, 71.37, -37.803, 5.247, -33.678, -4.37]
  Call Extruder 0.00929
  MoveL (T15485) to (112.64, 107.46, 16.9) mm, rotated rx 180 ry 0 rz -180 deg; joints [2.907, 71.37, -37.803, 5.247, -33.678, -4.37]
  Call Extruder 0.18127
  MoveL (T15486) to (107.78, 112.32, 16.9) mm, rotated rx 180 ry 0 rz -180 deg; joints [2.907, 71.37, -37.803, 5.247, -33.678, -4.37]
  Call Extruder 0.00976
  MoveL (T15487) to (107.61, 111.99, 16.9) mm, rotated rx 180 ry 0 rz -180 deg; joints [2.907, 71.37, -37.803, 5.247, -33.678, -4.37]
  Call Extruder 0.17825
  MoveL (T15488) to (112.39, 107.21, 16.9) mm, rotated rx 180 ry 0 rz -180 deg; joints [2.968, 71.379, -37.82, 5.358, -33.675, -4.463]
  Call Extruder 0.00765
  MoveL (T15489) to (112.18, 107, 16.9) mm, rotated rx 180 ry 0 rz -180 deg; joints [2.968, 71.379, -37.82, 5.358, -33.675, -4.463]
  Call Extruder 0.03908
  MoveL (T15490) to (111.14, 108.05, 16.9) mm, rotated rx 180 ry 0 rz -180 deg; joints [2.968, 71.379, -37.82, 5.358, -33.675, -4.463]
  Call Extruder 0.00424
  MoveL (T15491) to (110.99, 108.11, 16.9) mm, rotated rx 180 ry 0 rz -180 deg; joints [1.435, 66.932, -29.455, 2.358, -37.5, -1.871]
  Call Extruder 0.13224
  MoveL (T15492) to (107.44, 111.66, 16.9) mm, rotated rx 180 ry 0 rz -180 deg; joints [1.435, 66.932, -29.455, 2.358, -37.5, -1.871]
  Call Extruder 0.00976
  MoveL (T15493) to (107.27, 111.33, 16.9) mm, rotated rx 180 ry 0 rz -180 deg; joints [1.435, 66.932, -29.455, 2.358, -37.5, -1.871]
  Call Extruder 0.11932
  MoveL (T15494) to (110.47, 108.13, 16.9) mm, rotated rx 180 ry 0 rz -180 deg; joints [1.437, 66.78, -29.17, 2.354, -37.633, -1.864]
  Call Extruder 0.01314
  MoveL (T15495) to (109.97, 108.13, 16.9) mm, rotated rx 180 ry 0 rz -180 deg; joints [1.437, 66.78, -29.17, 2.354, -37.633, -1.864]
  Call Extruder 0.10702
  MoveL (T15496) to (107.1, 111, 16.9) mm, rotated rx 180 ry 0 rz -180 deg; joints [1.437, 66.78, -29.17, 2.354, -37.633, -1.864]
  Call Extruder 0.00976
  MoveL (T15497) to (106.93, 110.67, 16.9) mm, rotated rx 180 ry 0 rz -180 deg; joints [3.029, 71.389, -37.838, 5.469, -33.671, -4.555]
  Call Extruder 0.09471
  MoveL (T15498) to (109.47, 108.13, 16.9) mm, rotated rx 180 ry 0 rz -180 deg; joints [3.029, 71.389, -37.838, 5.469, -33.671, -4.555]
  Call Extruder 0.01314
  MoveL (T15499) to (108.98, 108.13, 16.9) mm, rotated rx 180 ry 0 rz -180 deg; joints [3.029, 71.389, -37.838, 5.469, -33.671, -4.555]
  Call Extruder 0.08241
  MoveL (T15500) to (106.77, 110.34, 16.9) mm, rotated rx 180 ry 0 rz -180 deg; joints [3.09, 71.399, -37.857, 5.579, -33.667, -4.648]
  Call Extruder 0.00976
  MoveL (T15501) to (106.6, 110.01, 16.9) mm, rotated rx 180 ry 0 rz -180 deg; joints [3.09, 71.399, -37.857, 5.579, -33.667, -4.648]
  Call Extruder 0.07011
  MoveL (T15502) to (108.48, 108.13, 16.9) mm, rotated rx 180 ry 0 rz -180 deg; joints [3.09, 71.399, -37.857, 5.579, -33.667, -4.648]
  Call Extruder 0.01314
  MoveL (T15503) to (107.98, 108.13, 16.9) mm, rotated rx 180 ry 0 rz -180 deg; joints [1.439, 66.629, -28.886, 2.349, -37.766, -1.858]
  Call Extruder 0.05781
  MoveL (T15504) to (106.43, 109.68, 16.9) mm, rotated rx 180 ry 0 rz -180 deg; joints [1.439, 66.629, -28.886, 2.349, -37.766, -1.858]
  Call Extruder 0.00976
  MoveL (T15505) to (106.26, 109.35, 16.9) mm, rotated rx 180 ry 0 rz -180 deg; joints [1.44, 66.479, -28.604, 2.345, -37.898, -1.851]
  Call Extruder 0.04551
  MoveL (T15506) to (107.48, 108.13, 16.9) mm, rotated rx 180 ry 0 rz -180 deg; joints [1.44, 66.479, -28.604, 2.345, -37.898, -1.851]
  Call Extruder 0.01314
  MoveL (T15507) to (106.98, 108.13, 16.9) mm, rotated rx 180 ry 0 rz -180 deg; joints [3.15, 71.409, -37.875, 5.69, -33.664, -4.741]
  Call Extruder 0.03321
  MoveL (T15508) to (106.09, 109.02, 16.9) mm, rotated rx 180 ry 0 rz -180 deg; joints [3.15, 71.409, -37.875, 5.69, -33.664, -4.741]
  Call Extruder 0.00976
  MoveL (T15509) to (105.92, 108.69, 16.9) mm, rotated rx 180 ry 0 rz -180 deg; joints [3.15, 71.409, -37.875, 5.69, -33.664, -4.741]
  Call Extruder 0.02091
  MoveL (T15510) to (106.48, 108.13, 16.9) mm, rotated rx 180 ry 0 rz -180 deg; joints [3.211, 71.419, -37.894, 5.801, -33.66, -4.833]
  Call Extruder 0.01314
  MoveL (T15511) to (105.99, 108.13, 16.9) mm, rotated rx 180 ry 0 rz -180 deg; joints [3.211, 71.419, -37.894, 5.801, -33.66, -4.833]
  Call Extruder 0.01292
  MoveL (T15512) to (105.64, 108.48, 16.9) mm, rotated rx 180 ry 0 rz -180 deg; joints [3.211, 71.419, -37.894, 5.801, -33.66, -4.833]
  Set speed (45.0 mm/s)
  Call Extruder -1.6
  MoveL (T15513) to (105.64, 108.48, 16.9) mm, rotated rx 180 ry 0 rz -180 deg; joints [1.442, 66.329, -28.323, 2.341, -38.029, -1.844]
  Set speed (120.0 mm/s)
  MoveL (T15514) to (105.64, 108.48, 16.9) mm, rotated rx 180 ry 0 rz -180 deg; joints [1.505, 66.333, -28.331, 2.443, -38.028, -1.925]
  Call Extruder -0.17462
  MoveL (T15515) to (105.99, 108.13, 16.9) mm, rotated rx 180 ry 0 rz -180 deg; joints [1.505, 66.333, -28.331, 2.443, -38.028, -1.925]
  Call Extruder -0.17749
  MoveL (T15516) to (106.48, 108.13, 16.9) mm, rotated rx 180 ry 0 rz -180 deg; joints [3.215, 71.236, -37.552, 5.782, -33.82, -4.809]
  Call Extruder -0.02788
  MoveL (T15517) to (106.43, 108.19, 16.9) mm, rotated rx 180 ry 0 rz -180 deg; joints [3.215, 71.236, -37.552, 5.782, -33.82, -4.809]
  Set speed (45.0 mm/s)
  Call Extruder -0.02
  MoveL (T15518) to (106.43, 108.19, 16.9) mm, rotated rx 180 ry 0 rz -180 deg; joints [3.218, 71.056, -37.212, 5.765, -33.979, -4.785]
  Set speed (150.0 mm/s)
  MoveL (T15519) to (106.43, 108.19, 18.9) mm, rotated rx 180 ry 0 rz -180 deg; joints [3.218, 71.056, -37.212, 5.765, -33.979, -4.785]
  MoveL (T15520) to (120.54, 120.54, 18.9) mm, rotated rx 180 ry 0 rz -180 deg; joints [1.568, 66.337, -28.338, 2.545, -38.027, -2.005]
  MoveL (T15521) to (120.54, 120.54, 16.9) mm, rotated rx 180 ry 0 rz -180 deg; joints [1.631, 66.341, -28.346, 2.648, -38.025, -2.086]
  Set speed (40.0 mm/s)
  Call Extruder 2.0
  MoveL (T15522) to (120.54, 120.54, 16.9) mm, rotated rx 180 ry 0 rz -180 deg; joints [1.631, 66.341, -28.346, 2.648, -38.025, -2.086]
  Set speed (50.0 mm/s)
  MoveL (T15523) to (120.54, 120.54, 16.9) mm, rotated rx 180 ry 0 rz -180 deg; joints [3.222, 70.876, -36.874, 5.747, -34.136, -4.762]
  Call Extruder 0.02637
  MoveL (T15524) to (121.16, 121.16, 16.9) mm, rotated rx 180 ry 0 rz -180 deg; joints [3.225, 70.699, -36.54, 5.73, -34.292, -4.739]
  Set speed (45.0 mm/s)
  Call Extruder -1.6
  MoveL (T15525) to (121.16, 121.16, 16.9) mm, rotated rx 180 ry 0 rz -180 deg; joints [3.225, 70.699, -36.54, 5.73, -34.292, -4.739]
  Set speed (120.0 mm/s)
  MoveL (T15526) to (121.16, 121.16, 16.9) mm, rotated rx 180 ry 0 rz -180 deg; joints [1.694, 66.346, -28.354, 2.75, -38.024, -2.167]
  Call Extruder -0.30841
  MoveL (T15527) to (120.54, 120.54, 16.9) mm, rotated rx 180 ry 0 rz -180 deg; joints [1.694, 66.346, -28.354, 2.75, -38.024, -2.167]
  Set speed (45.0 mm/s)
  Call Extruder -0.09159
  MoveL (T15528) to (120.54, 120.54, 16.9) mm, rotated rx 180 ry 0 rz -180 deg; joints [1.694, 66.346, -28.354, 2.75, -38.024, -2.167]
  Set speed (150.0 mm/s)
  MoveL (T15529) to (120.54, 120.54, 18.9) mm, rotated rx 180 ry 0 rz -180 deg; joints [1.757, 66.35, -28.362, 2.852, -38.022, -2.248]
  MoveL (T15530) to (104.34, 103.54, 18.9) mm, rotated rx 180 ry 0 rz -180 deg; joints [1.757, 66.35, -28.362, 2.852, -38.022, -2.248]
  MoveL (T15531) to (104.34, 103.54, 17.1) mm, rotated rx 180 ry 0 rz -180 deg; joints [1.757, 66.35, -28.362, 2.852, -38.022, -2.248]
  Set speed (40.0 mm/s)
  Call Extruder 2.0
  MoveL (T15532) to (104.34, 103.54, 17.1) mm, rotated rx 180 ry 0 rz -180 deg; joints [3.228, 70.522, -36.208, 5.714, -34.447, -4.717]
  Call Extruder 0.52159
  MoveL (T15533) to (121.46, 103.54, 17.1) mm, rotated rx 180 ry 0 rz -180 deg; joints [3.228, 70.522, -36.208, 5.714, -34.447, -4.717]
  Call Extruder 0.54596
  MoveL (T15534) to (121.46, 121.46, 17.1) mm, rotated rx 180 ry 0 rz -180 deg; joints [3.228, 70.522, -36.208, 5.714, -34.447, -4.717]
  Call Extruder 0.54596
  MoveL (T15535) to (103.54, 121.46, 17.1) mm, rotated rx 180 ry 0 rz -180 deg; joints [3.228, 70.522, -36.208, 5.714, -34.447, -4.717]
  Call Extruder 0.54596
  MoveL (T15536) to (103.54, 103.54, 17.1) mm, rotated rx 180 ry 0 rz -180 deg; joints [3.232, 70.347, -35.878, 5.698, -34.601, -4.695]
  Call Extruder 0.02254
  MoveL (T15537) to (104.28, 103.54, 17.1) mm, rotated rx 180 ry 0 rz -180 deg; joints [3.232, 70.347, -35.878, 5.698, -34.601, -4.695]
  Set speed (150.0 mm/s)
  MoveL (T15538) to (103.53, 103.13, 17.1) mm, rotated rx 180 ry 0 rz -180 deg; joints [1.82, 66.355, -28.371, 2.955, -38.021, -2.329]
  Set speed (40.0 mm/s)
  MoveL (T15539) to (103.53, 103.13, 17.1) mm, rotated rx 180 ry 0 rz -180 deg; joints [1.882, 66.36, -28.38, 3.057, -38.019, -2.409]
  Call Extruder 0.55858
  MoveL (T15540) to (121.87, 103.13, 17.1) mm, rotated rx 180 ry 0 rz -180 deg; joints [1.882, 66.36, -28.38, 3.057, -38.019, -2.409]
  Call Extruder 0.57077
  MoveL (T15541) to (121.87, 121.87, 17.1) mm, rotated rx 180 ry 0 rz -180 deg; joints [1.882, 66.36, -28.38, 3.057, -38.019, -2.409]
  Call Extruder 0.57077
  MoveL (T15542) to (103.13, 121.87, 17.1) mm, rotated rx 180 ry 0 rz -180 deg; joints [3.235, 70.173, -35.552, 5.682, -34.754, -4.673]
  Call Extruder 0.57077
  MoveL (T15543) to (103.13, 103.13, 17.1) mm, rotated rx 180 ry 0 rz -180 deg; joints [3.235, 70.173, -35.552, 5.682, -34.754, -4.673]
  Call Extruder 0.01036
  MoveL (T15544) to (103.47, 103.13, 17.1) mm, rotated rx 180 ry 0 rz -180 deg; joints [3.239, 70.001, -35.227, 5.666, -34.905, -4.652]
  Set speed (150.0 mm/s)
  MoveL (T15545) to (102.72, 102.81, 17.1) mm, rotated rx 180 ry 0 rz -180 deg; joints [3.239, 70.001, -35.227, 5.666, -34.905, -4.652]
  Set speed (25.0 mm/s)
  MoveL (T15546) to (102.72, 102.81, 17.1) mm, rotated rx 180 ry 0 rz -180 deg; joints [3.239, 70.001, -35.227, 5.666, -34.905, -4.652]
  Call Extruder 0.00259
  MoveL (T15547) to (102.72, 102.72, 17.1) mm, rotated rx 180 ry 0 rz -180 deg; joints [1.945, 66.365, -28.39, 3.16, -38.017, -2.49]
  Call Extruder 0.59557
  MoveL (T15548) to (122.28, 102.72, 17.1) mm, rotated rx 180 ry 0 rz -180 deg; joints [1.945, 66.365, -28.39, 3.16, -38.017, -2.49]
  Call Extruder 0.59557
  MoveL (T15549) to (122.28, 122.28, 17.1) mm, rotated rx 180 ry 0 rz -180 deg; joints [2.008, 66.37, -28.399, 3.262, -38.016, -2.571]
  Call Extruder 0.59557
  MoveL (T15550) to (102.72, 122.28, 17.1) mm, rotated rx 180 ry 0 rz -180 deg; joints [2.008, 66.37, -28.399, 3.262, -38.016, -2.571]
  Call Extruder 0.59115
  MoveL (T15551) to (102.72, 102.87, 17.1) mm, rotated rx 180 ry 0 rz -180 deg; joints [3.242, 69.83, -34.905, 5.651, -35.055, -4.631]
  Set speed (150.0 mm/s)
  MoveL (T15552) to (102.78, 102.75, 17.1) mm, rotated rx 180 ry 0 rz -180 deg; joints [3.246, 69.66, -34.586, 5.636, -35.205, -4.61]
  Set speed (45.0 mm/s)
  Call Extruder -1.6
  MoveL (T15553) to (102.78, 102.75, 17.1) mm, rotated rx 180 ry 0 rz -180 deg; joints [3.246, 69.66, -34.586, 5.636, -35.205, -4.61]
  Set speed (120.0 mm/s)
  MoveL (T15554) to (102.78, 102.75, 17.1) mm, rotated rx 180 ry 0 rz -180 deg; joints [2.071, 66.375, -28.409, 3.365, -38.014, -2.652]
  Call Extruder -0.05166
  MoveL (T15555) to (102.72, 102.72, 17.1) mm, rotated rx 180 ry 0 rz -180 deg; joints [2.134, 66.381, -28.42, 3.467, -38.012, -2.733]
  Call Extruder -0.32834
  MoveL (T15556) to (103.65, 102.72, 17.1) mm, rotated rx 180 ry 0 rz -180 deg; joints [2.134, 66.381, -28.42, 3.467, -38.012, -2.733]
  Set speed (45.0 mm/s)
  Call Extruder -0.02
  MoveL (T15557) to (103.65, 102.72, 17.1) mm, rotated rx 180 ry 0 rz -180 deg; joints [3.249, 69.491, -34.268, 5.622, -35.353, -4.59]
  Set speed (150.0 mm/s)
  MoveL (T15558) to (103.65, 102.72, 19.1) mm, rotated rx 180 ry 0 rz -180 deg; joints [3.249, 69.491, -34.268, 5.622, -35.353, -4.59]
  MoveL (T15559) to (106.08, 103.93, 19.1) mm, rotated rx 180 ry 0 rz -180 deg; joints [3.249, 69.491, -34.268, 5.622, -35.353, -4.59]
  MoveL (T15560) to (106.08, 103.93, 17.1) mm, rotated rx 180 ry 0 rz -180 deg; joints [3.253, 69.323, -33.953, 5.607, -35.5, -4.57]
  Set speed (40.0 mm/s)
  Call Extruder 2.0
  MoveL (T15561) to (106.08, 103.93, 17.1) mm, rotated rx 180 ry 0 rz -180 deg; joints [3.253, 69.323, -33.953, 5.607, -35.5, -4.57]
  Set speed (50.0 mm/s)
  MoveL (T15562) to (106.08, 103.93, 17.1) mm, rotated rx 180 ry 0 rz -180 deg; joints [3.253, 69.323, -33.953, 5.607, -35.5, -4.57]
  Call Extruder 0.00361
  MoveL (T15563) to (106.17, 103.84, 17.1) mm, rotated rx 180 ry 0 rz -180 deg; joints [2.197, 66.386, -28.43, 3.57, -38.01, -2.814]
  Call Extruder 0.0708
  MoveL (T15564) to (103.84, 103.84, 17.1) mm, rotated rx 180 ry 0 rz -180 deg; joints [2.197, 66.386, -28.43, 3.57, -38.01, -2.814]
  Call Extruder 0.05255
  MoveL (T15565) to (105.06, 105.06, 17.1) mm, rotated rx 180 ry 0 rz -180 deg; joints [2.197, 66.386, -28.43, 3.57, -38.01, -2.814]
  Call Extruder 0.03217
  MoveL (T15566) to (105.06, 106.12, 17.1) mm, rotated rx 180 ry 0 rz -180 deg; joints [2.26, 66.392, -28.441, 3.672, -38.008, -2.895]
  Call Extruder 0.0525
  MoveL (T15567) to (103.84, 107.34, 17.1) mm, rotated rx 180 ry 0 rz -180 deg; joints [2.26, 66.392, -28.441, 3.672, -38.008, -2.895]
  Call Extruder 0.03385
  MoveL (T15568) to (103.84, 108.45, 17.1) mm, rotated rx 180 ry 0 rz -180 deg; joints [2.26, 66.392, -28.441, 3.672, -38.008, -2.895]
  Call Extruder 0.13495
  MoveL (T15569) to (106.98, 111.58, 17.1) mm, rotated rx 180 ry 0 rz -180 deg; joints [3.256, 69.157, -33.64, 5.593, -35.646, -4.55]
  Call Extruder 0.04156
  MoveL (T15570) to (107.6, 112.8, 17.1) mm, rotated rx 180 ry 0 rz -180 deg; joints [3.256, 69.157, -33.64, 5.593, -35.646, -4.55]
  Call Extruder 0.16166
  MoveL (T15571) to (103.84, 116.55, 17.1) mm, rotated rx 180 ry 0 rz -180 deg; joints [3.26, 68.992, -33.33, 5.58, -35.791, -4.531]
  Call Extruder 0.03385
  MoveL (T15572) to (103.84, 117.66, 17.1) mm, rotated rx 180 ry 0 rz -180 deg; joints [3.26, 68.992, -33.33, 5.58, -35.791, -4.531]
  Call Extruder 0.05612
  MoveL (T15573) to (105.15, 118.96, 17.1) mm, rotated rx 180 ry 0 rz -180 deg; joints [3.26, 68.992, -33.33, 5.58, -35.791, -4.531]
  Call Extruder 0.02709
  MoveL (T15574) to (105.15, 119.85, 17.1) mm, rotated rx 180 ry 0 rz -180 deg; joints [2.323, 66.398, -28.452, 3.774, -38.006, -2.976]
  Call Extruder 0.05612
  MoveL (T15575) to (103.84, 121.16, 17.1) mm, rotated rx 180 ry 0 rz -180 deg; joints [2.323, 66.398, -28.452, 3.774, -38.006, -2.976]
  Call Extruder 0.06345
  MoveL (T15576) to (105.93, 121.16, 17.1) mm, rotated rx 180 ry 0 rz -180 deg; joints [2.323, 66.398, -28.452, 3.774, -38.006, -2.976]
  Call Extruder 0.01096
  MoveL (T15577) to (105.67, 120.9, 17.1) mm, rotated rx 180 ry 0 rz -180 deg; joints [2.386, 66.404, -28.464, 3.877, -38.004, -3.057]
  Set speed (45.0 mm/s)
  Call Extruder -1.6
  MoveL (T15578) to (105.67, 120.9, 17.1) mm, rotated rx 180 ry 0 rz -180 deg; joints [3.263, 68.828, -33.021, 5.566, -35.935, -4.512]
  Set speed (120.0 mm/s)
  MoveL (T15579) to (105.67, 120.9, 17.1) mm, rotated rx 180 ry 0 rz -180 deg; joints [3.263, 68.828, -33.021, 5.566, -35.935, -4.512]
  Call Extruder -0.12811
  MoveL (T15580) to (105.93, 121.16, 17.1) mm, rotated rx 180 ry 0 rz -180 deg; joints [3.267, 68.665, -32.714, 5.553, -36.079, -4.493]
  Call Extruder -0.25189
  MoveL (T15581) to (105.22, 121.16, 17.1) mm, rotated rx 180 ry 0 rz -180 deg; joints [3.267, 68.665, -32.714, 5.553, -36.079, -4.493]
  Set speed (45.0 mm/s)
  Call Extruder -0.02
  MoveL (T15582) to (105.22, 121.16, 17.1) mm, rotated rx 180 ry 0 rz -180 deg; joints [2.449, 66.41, -28.476, 3.979, -38.002, -3.138]
  Set speed (150.0 mm/s)
  MoveL (T15583) to (105.22, 121.16, 19.1) mm, rotated rx 180 ry 0 rz -180 deg; joints [2.449, 66.41, -28.476, 3.979, -38.002, -3.138]
  MoveL (T15584) to (105.15, 117.23, 19.1) mm, rotated rx 180 ry 0 rz -180 deg; joints [2.512, 66.417, -28.488, 4.082, -38, -3.219]
  MoveL (T15585) to (105.15, 117.23, 17.1) mm, rotated rx 180 ry 0 rz -180 deg; joints [2.512, 66.417, -28.488, 4.082, -38, -3.219]
  Set speed (40.0 mm/s)
  Call Extruder 2.0
  MoveL (T15586) to (105.15, 117.23, 17.1) mm, rotated rx 180 ry 0 rz -180 deg; joints [2.512, 66.417, -28.488, 4.082, -38, -3.219]
  Set speed (50.0 mm/s)
  MoveL (T15587) to (105.15, 117.23, 17.1) mm, rotated rx 180 ry 0 rz -180 deg; joints [3.27, 68.503, -32.41, 5.54, -36.221, -4.474]
  Call Extruder 0.04143
  MoveL (T15588) to (105.15, 115.87, 17.1) mm, rotated rx 180 ry 0 rz -180 deg; joints [3.27, 68.503, -32.41, 5.54, -36.221, -4.474]
  Call Extruder 0.00661
  MoveL (T15589) to (105.23, 115.67, 17.1) mm, rotated rx 180 ry 0 rz -180 deg; joints [3.274, 68.342, -32.107, 5.527, -36.362, -4.456]
  Call Extruder 0.02637
  MoveL (T15590) to (105.84, 115.05, 17.1) mm, rotated rx 180 ry 0 rz -180 deg; joints [3.274, 68.342, -32.107, 5.527, -36.362, -4.456]
  Call Extruder 0.08606
  MoveL (T15591) to (103.84, 113.06, 17.1) mm, rotated rx 180 ry 0 rz -180 deg; joints [3.274, 68.342, -32.107, 5.527, -36.362, -4.456]
  Call Extruder 0.03385
  MoveL (T15592) to (103.84, 111.94, 17.1) mm, rotated rx 180 ry 0 rz -180 deg; joints [3.274, 68.342, -32.107, 5.527, -36.362, -4.456]
  Call Extruder 0.09463
  MoveL (T15593) to (106.04, 109.75, 17.1) mm, rotated rx 180 ry 0 rz -180 deg; joints [2.575, 66.424, -28.5, 4.184, -37.997, -3.3]
  Call Extruder 0.05062
  MoveL (T15594) to (105.29, 108.27, 17.1) mm, rotated rx 180 ry 0 rz -180 deg; joints [2.575, 66.424, -28.5, 4.184, -37.997, -3.3]
  Call Extruder 0.02377
  MoveL (T15595) to (105.1, 107.51, 17.1) mm, rotated rx 180 ry 0 rz -180 deg; joints [2.575, 66.424, -28.5, 4.184, -37.997, -3.3]
  Set speed (45.0 mm/s)
  Call Extruder -1.6
  MoveL (T15596) to (105.1, 107.51, 17.1) mm, rotated rx 180 ry 0 rz -180 deg; joints [2.638, 66.43, -28.513, 4.287, -37.995, -3.381]
  Set speed (120.0 mm/s)
  MoveL (T15597) to (105.1, 107.51, 17.1) mm, rotated rx 180 ry 0 rz -180 deg; joints [3.277, 68.182, -31.806, 5.515, -36.503, -4.438]
  Call Extruder -0.278
  MoveL (T15598) to (105.29, 108.27, 17.1) mm, rotated rx 180 ry 0 rz -180 deg; joints [3.277, 68.182, -31.806, 5.515, -36.503, -4.438]
  Call Extruder -0.102
  MoveL (T15599) to (105.42, 108.52, 17.1) mm, rotated rx 180 ry 0 rz -180 deg; joints [3.281, 68.023, -31.507, 5.503, -36.642, -4.42]
  Set speed (45.0 mm/s)
  Call Extruder -0.02
  MoveL (T15600) to (105.42, 108.52, 17.1) mm, rotated rx 180 ry 0 rz -180 deg; joints [3.281, 68.023, -31.507, 5.503, -36.642, -4.42]
  Set speed (150.0 mm/s)
  MoveL (T15601) to (105.42, 108.52, 19.1) mm, rotated rx 180 ry 0 rz -180 deg; joints [2.7, 66.437, -28.526, 4.39, -37.993, -3.462]
  MoveL (T15602) to (119.44, 110.51, 19.1) mm, rotated rx 180 ry 0 rz -180 deg; joints [2.7, 66.437, -28.526, 4.39, -37.993, -3.462]
  MoveL (T15603) to (119.44, 110.51, 17.1) mm, rotated rx 180 ry 0 rz -180 deg; joints [2.763, 66.444, -28.54, 4.492, -37.99, -3.543]
  Set speed (40.0 mm/s)
  Call Extruder 2.0
  MoveL (T15604) to (119.44, 110.51, 17.1) mm, rotated rx 180 ry 0 rz -180 deg; joints [2.763, 66.444, -28.54, 4.492, -37.99, -3.543]
  Set speed (50.0 mm/s)
  MoveL (T15605) to (119.44, 110.51, 17.1) mm, rotated rx 180 ry 0 rz -180 deg; joints [3.285, 67.865, -31.21, 5.491, -36.781, -4.403]
  Call Extruder 0.05098
  MoveL (T15606) to (118.25, 111.7, 17.1) mm, rotated rx 180 ry 0 rz -180 deg; joints [3.285, 67.865, -31.21, 5.491, -36.781, -4.403]
  Call Extruder 0.00661
  MoveL (T15607) to (118.05, 111.78, 17.1) mm, rotated rx 180 ry 0 rz -180 deg; joints [3.288, 67.708, -30.915, 5.479, -36.919, -4.385]
  Call Extruder 0.00686
  MoveL (T15608) to (117.83, 111.78, 17.1) mm, rotated rx 180 ry 0 rz -180 deg; joints [2.826, 66.452, -28.553, 4.595, -37.988, -3.624]
  Call Extruder 0.01607
  MoveL (T15609) to (117.45, 112.15, 17.1) mm, rotated rx 180 ry 0 rz -180 deg; joints [2.826, 66.452, -28.553, 4.595, -37.988, -3.624]
  Call Extruder 0.01616
  MoveL (T15610) to (117.69, 112.62, 17.1) mm, rotated rx 180 ry 0 rz -180 deg; joints [2.826, 66.452, -28.553, 4.595, -37.988, -3.624]
  Call Extruder 0.05338
  MoveL (T15611) to (118.94, 111.39, 17.1) mm, rotated rx 180 ry 0 rz -180 deg; joints [2.889, 66.459, -28.567, 4.697, -37.985, -3.705]
  Call Extruder 0.00661
  MoveL (T15612) to (119.14, 111.3, 17.1) mm, rotated rx 180 ry 0 rz -180 deg; joints [3.292, 67.552, -30.621, 5.468, -37.056, -4.368]
  Call Extruder 0.04204
  MoveL (T15613) to (120.52, 111.31, 17.1) mm, rotated rx 180 ry 0 rz -180 deg; joints [3.292, 67.552, -30.621, 5.468, -37.056, -4.368]
  Call Extruder 0.04035
  MoveL (T15614) to (119.58, 110.37, 17.1) mm, rotated rx 180 ry 0 rz -180 deg; joints [3.292, 67.552, -30.621, 5.468, -37.056, -4.368]
  Call Extruder 0.03053
  MoveL (T15615) to (120.29, 109.66, 17.1) mm, rotated rx 180 ry 0 rz -180 deg; joints [3.295, 67.397, -30.33, 5.457, -37.192, -4.352]
  Call Extruder 0.00661
  MoveL (T15616) to (120.37, 109.46, 17.1) mm, rotated rx 180 ry 0 rz -180 deg; joints [3.295, 67.397, -30.33, 5.457, -37.192, -4.352]
  Call Extruder 0.00686
  MoveL (T15617) to (120.37, 109.23, 17.1) mm, rotated rx 180 ry 0 rz -180 deg; joints [2.952, 66.467, -28.582, 4.8, -37.983, -3.787]
  Call Extruder 0.03378
  MoveL (T15618) to (121.16, 108.45, 17.1) mm, rotated rx 180 ry 0 rz -180 deg; joints [2.952, 66.467, -28.582, 4.8, -37.983, -3.787]
  Call Extruder 0.03385
  MoveL (T15619) to (121.16, 107.34, 17.1) mm, rotated rx 180 ry 0 rz -180 deg; joints [3.015, 66.475, -28.596, 4.903, -37.98, -3.868]
  Call Extruder 0.03378
  MoveL (T15620) to (120.37, 106.56, 17.1) mm, rotated rx 180 ry 0 rz -180 deg; joints [3.015, 66.475, -28.596, 4.903, -37.98, -3.868]
  Call Extruder 0.04531
  MoveL (T15621) to (120.37, 105.07, 17.1) mm, rotated rx 180 ry 0 rz -180 deg; joints [3.015, 66.475, -28.596, 4.903, -37.98, -3.868]
  Call Extruder 0.00661
  MoveL (T15622) to (120.29, 104.87, 17.1) mm, rotated rx 180 ry 0 rz -180 deg; joints [3.299, 67.242, -30.04, 5.446, -37.328, -4.335]
  Call Extruder 0.00334
  MoveL (T15623) to (120.21, 104.79, 17.1) mm, rotated rx 180 ry 0 rz -180 deg; joints [3.299, 67.242, -30.04, 5.446, -37.328, -4.335]
  Call Extruder 0.04071
  MoveL (T15624) to (121.16, 103.84, 17.1) mm, rotated rx 180 ry 0 rz -180 deg; joints [3.302, 67.089, -29.752, 5.435, -37.462, -4.319]
  Call Extruder 0.07441
  MoveL (T15625) to (121.16, 106.29, 17.1) mm, rotated rx 180 ry 0 rz -180 deg; joints [3.302, 67.089, -29.752, 5.435, -37.462, -4.319]
  Set speed (150.0 mm/s)
  MoveL (T15626) to (120.15, 105.3, 17.1) mm, rotated rx 180 ry 0 rz -180 deg; joints [3.14, 66.491, -28.626, 5.108, -37.975, -4.03]
  Set speed (40.0 mm/s)
  MoveL (T15627) to (120.15, 105.3, 17.1) mm, rotated rx 180 ry 0 rz -180 deg; joints [3.14, 66.491, -28.626, 5.108, -37.975, -4.03]
  Call Extruder 0.06313
  MoveL (T15628) to (118.69, 103.84, 17.1) mm, rotated rx 180 ry 0 rz -180 deg; joints [3.14, 66.491, -28.626, 5.108, -37.975, -4.03]
  Call Extruder 0.0177
  MoveL (T15629) to (118.11, 103.84, 17.1) mm, rotated rx 180 ry 0 rz -180 deg; joints [3.14, 66.491, -28.626, 5.108, -37.975, -4.03]
  Call Extruder 0.08024
  MoveL (T15630) to (119.96, 105.7, 17.1) mm, rotated rx 180 ry 0 rz -180 deg; joints [3.306, 66.937, -29.465, 5.424, -37.596, -4.303]
  Call Extruder 0.0177
  MoveL (T15631) to (119.96, 106.28, 17.1) mm, rotated rx 180 ry 0 rz -180 deg; joints [3.31, 66.785, -29.18, 5.414, -37.729, -4.287]
  Call Extruder 0.10527
  MoveL (T15632) to (117.53, 103.84, 17.1) mm, rotated rx 180 ry 0 rz -180 deg; joints [3.31, 66.785, -29.18, 5.414, -37.729, -4.287]
  Call Extruder 0.0177
  MoveL (T15633) to (116.95, 103.84, 17.1) mm, rotated rx 180 ry 0 rz -180 deg; joints [3.203, 66.499, -28.642, 5.211, -37.972, -4.112]
  Call Extruder 0.1303
  MoveL (T15634) to (119.96, 106.86, 17.1) mm, rotated rx 180 ry 0 rz -180 deg; joints [3.203, 66.499, -28.642, 5.211, -37.972, -4.112]
  Call Extruder 0.0177
  MoveL (T15635) to (119.96, 107.43, 17.1) mm, rotated rx 180 ry 0 rz -180 deg; joints [3.203, 66.499, -28.642, 5.211, -37.972, -4.112]
  Call Extruder 0.15533
  MoveL (T15636) to (116.38, 103.84, 17.1) mm, rotated rx 180 ry 0 rz -180 deg; joints [3.266, 66.507, -28.658, 5.313, -37.969, -4.193]
  Call Extruder 0.0177
  MoveL (T15637) to (115.8, 103.84, 17.1) mm, rotated rx 180 ry 0 rz -180 deg; joints [3.266, 66.507, -28.658, 5.313, -37.969, -4.193]
  Call Extruder 0.18036
  MoveL (T15638) to (119.96, 108.01, 17.1) mm, rotated rx 180 ry 0 rz -180 deg; joints [3.266, 66.507, -28.658, 5.313, -37.969, -4.193]
  Call Extruder 0.0177
  MoveL (T15639) to (119.96, 108.59, 17.1) mm, rotated rx 180 ry 0 rz -180 deg; joints [3.332, 66.685, -28.991, 5.439, -37.819, -4.302]
  Call Extruder 0.20539
  MoveL (T15640) to (115.22, 103.84, 17.1) mm, rotated rx 180 ry 0 rz -180 deg; joints [3.332, 66.685, -28.991, 5.439, -37.819, -4.302]
  Call Extruder 0.0177
  MoveL (T15641) to (114.64, 103.84, 17.1) mm, rotated rx 180 ry 0 rz -180 deg; joints [3.332, 66.685, -28.991, 5.439, -37.819, -4.302]
  Call Extruder 0.23042
  MoveL (T15642) to (119.96, 109.17, 17.1) mm, rotated rx 180 ry 0 rz -180 deg; joints [3.332, 66.685, -28.991, 5.439, -37.819, -4.302]
  Call Extruder 0.00643
  MoveL (T15643) to (119.96, 109.38, 17.1) mm, rotated rx 180 ry 0 rz -180 deg; joints [3.332, 66.685, -28.991, 5.439, -37.819, -4.302]
  Call Extruder 0.00169
  MoveL (T15644) to (119.94, 109.43, 17.1) mm, rotated rx 180 ry 0 rz -180 deg; joints [3.332, 66.685, -28.991, 5.439, -37.819, -4.302]
  Call Extruder 0.00641
  MoveL (T15645) to (119.8, 109.58, 17.1) mm, rotated rx 180 ry 0 rz -180 deg; joints [3.332, 66.685, -28.991, 5.439, -37.819, -4.302]
  Call Extruder 0.24813
  MoveL (T15646) to (114.06, 103.84, 17.1) mm, rotated rx 180 ry 0 rz -180 deg; joints [3.332, 66.685, -28.991, 5.439, -37.819, -4.302]
  Call Extruder 0.0177
  MoveL (T15647) to (113.48, 103.84, 17.1) mm, rotated rx 180 ry 0 rz -180 deg; joints [3.266, 66.507, -28.658, 5.313, -37.969, -4.193]
  Call Extruder 0.26064
  MoveL (T15648) to (119.51, 109.87, 17.1) mm, rotated rx 180 ry 0 rz -180 deg; joints [3.266, 66.507, -28.658, 5.313, -37.969, -4.193]
  Call Extruder 0.01252
  MoveL (T15649) to (119.22, 110.16, 17.1) mm, rotated rx 180 ry 0 rz -180 deg; joints [3.266, 66.507, -28.658, 5.313, -37.969, -4.193]
  Call Extruder 0.27316
  MoveL (T15650) to (112.91, 103.84, 17.1) mm, rotated rx 180 ry 0 rz -180 deg; joints [3.25, 66.505, -28.654, 5.287, -37.97, -4.172]
  Call Extruder 0.0177
  MoveL (T15651) to (112.33, 103.84, 17.1) mm, rotated rx 180 ry 0 rz -180 deg; joints [3.25, 66.505, -28.654, 5.287, -37.97, -4.172]
  Call Extruder 0.28567
  MoveL (T15652) to (118.93, 110.44, 17.1) mm, rotated rx 180 ry 0 rz -180 deg; joints [3.25, 66.505, -28.654, 5.287, -37.97, -4.172]
  Call Extruder 0.01252
  MoveL (T15653) to (118.64, 110.73, 17.1) mm, rotated rx 180 ry 0 rz -180 deg; joints [3.25, 66.505, -28.654, 5.287, -37.97, -4.172]
  Call Extruder 0.29819
  MoveL (T15654) to (111.75, 103.84, 17.1) mm, rotated rx 180 ry 0 rz -180 deg; joints [3.25, 66.505, -28.654, 5.287, -37.97, -4.172]
  Call Extruder 0.0177
  MoveL (T15655) to (111.17, 103.84, 17.1) mm, rotated rx 180 ry 0 rz -180 deg; joints [3.25, 66.505, -28.654, 5.287, -37.97, -4.172]
  Call Extruder 0.3107
  MoveL (T15656) to (118.35, 111.02, 17.1) mm, rotated rx 180 ry 0 rz -180 deg; joints [3.25, 66.505, -28.654, 5.287, -37.97, -4.172]
  Call Extruder 0.01252
  MoveL (T15657) to (118.06, 111.31, 17.1) mm, rotated rx 180 ry 0 rz -180 deg; joints [3.25, 66.268, -28.615, 5.31, -37.772, -4.202]
  Call Extruder 0.32322
  MoveL (T15658) to (110.59, 103.84, 17.1) mm, rotated rx 180 ry 0 rz -180 deg; joints [1.407, 66.217, -28.52, 2.301, -37.72, -1.82]
  Call Extruder 0.0177
  MoveL (T15659) to (110.01, 103.84, 17.1) mm, rotated rx 180 ry 0 rz -180 deg; joints [1.407, 66.431, -28.555, 2.291, -37.898, -1.809]
  Call Extruder 0.32579
  MoveL (T15660) to (117.54, 111.37, 17.1) mm, rotated rx 180 ry 0 rz -180 deg; joints [1.407, 66.431, -28.555, 2.291, -37.898, -1.809]
  Call Extruder 0.0177
  MoveL (T15661) to (116.96, 111.37, 17.1) mm, rotated rx 180 ry 0 rz -180 deg; joints [1.407, 66.431, -28.555, 2.291, -37.898, -1.809]
  Call Extruder 0.32579
  MoveL (T15662) to (109.44, 103.84, 17.1) mm, rotated rx 180 ry 0 rz -180 deg; joints [1.407, 66.431, -28.555, 2.291, -37.898, -1.809]
  Call Extruder 0.0177
  MoveL (T15663) to (108.86, 103.84, 17.1) mm, rotated rx 180 ry 0 rz -180 deg; joints [1.407, 66.431, -28.555, 2.291, -37.898, -1.809]
  Call Extruder 0.36291
  MoveL (T15664) to (117.24, 112.23, 17.1) mm, rotated rx 180 ry 0 rz -180 deg; joints [1.407, 66.431, -28.555, 2.291, -37.898, -1.809]
  Set speed (45.0 mm/s)
  Call Extruder -1.6
  MoveL (T15665) to (117.24, 112.23, 17.1) mm, rotated rx 180 ry 0 rz -180 deg; joints [1.407, 66.431, -28.555, 2.291, -37.898, -1.809]
  Set speed (120.0 mm/s)
  MoveL (T15666) to (117.24, 112.23, 17.1) mm, rotated rx 180 ry 0 rz -180 deg; joints [1.407, 66.431, -28.555, 2.291, -37.898, -1.809]
  Call Extruder -0.38
  MoveL (T15667) to (116.49, 111.47, 17.1) mm, rotated rx 180 ry 0 rz -180 deg; joints [1.363, 71.27, -37.654, 2.461, -33.64, -2.049]
  Set speed (45.0 mm/s)
  Call Extruder -0.02
  MoveL (T15668) to (116.49, 111.47, 17.1) mm, rotated rx 180 ry 0 rz -180 deg; joints [1.363, 71.27, -37.654, 2.461, -33.64, -2.049]
  Set speed (150.0 mm/s)
  MoveL (T15669) to (116.49, 111.47, 19.1) mm, rotated rx 180 ry 0 rz -180 deg; joints [3.241, 71.497, -38.081, 5.871, -33.555, -4.898]
  MoveL (T15670) to (120.59, 111.53, 19.1) mm, rotated rx 180 ry 0 rz -180 deg; joints [3.241, 71.497, -38.081, 5.871, -33.555, -4.898]
  MoveL (T15671) to (120.59, 111.53, 17.1) mm, rotated rx 180 ry 0 rz -180 deg; joints [3.351, 66.417, -28.528, 5.447, -38.014, -4.296]
  Set speed (40.0 mm/s)
  Call Extruder 2.0
  MoveL (T15672) to (120.59, 111.53, 17.1) mm, rotated rx 180 ry 0 rz -180 deg; joints [3.351, 66.417, -28.528, 5.447, -38.014, -4.296]
  Call Extruder 0.02448
  MoveL (T15673) to (121.16, 112.09, 17.1) mm, rotated rx 180 ry 0 rz -180 deg; joints [3.351, 66.417, -28.528, 5.447, -38.014, -4.296]
  Call Extruder 0.0177
  MoveL (T15674) to (121.16, 112.67, 17.1) mm, rotated rx 180 ry 0 rz -180 deg; joints [1.409, 66.226, -28.169, 2.286, -38.079, -1.8]
  Call Extruder 0.0416
  MoveL (T15675) to (120.19, 111.71, 17.1) mm, rotated rx 180 ry 0 rz -180 deg; joints [1.409, 66.226, -28.169, 2.286, -38.079, -1.8]
  Call Extruder 0.01772
  MoveL (T15676) to (119.61, 111.71, 17.1) mm, rotated rx 180 ry 0 rz -180 deg; joints [1.407, 66.415, -28.526, 2.291, -37.912, -1.808]
  Call Extruder 0.06667
  MoveL (T15677) to (121.16, 113.25, 17.1) mm, rotated rx 180 ry 0 rz -180 deg; joints [1.407, 66.415, -28.526, 2.291, -37.912, -1.808]
  Call Extruder 0.0177
  MoveL (T15678) to (121.16, 113.83, 17.1) mm, rotated rx 180 ry 0 rz -180 deg; joints [1.407, 66.415, -28.526, 2.291, -37.912, -1.808]
  Call Extruder 0.08847
  MoveL (T15679) to (119.11, 111.79, 17.1) mm, rotated rx 180 ry 0 rz -180 deg; joints [1.365, 66.221, -28.161, 2.214, -38.081, -1.743]
  Call Extruder 0.01252
  MoveL (T15680) to (118.82, 112.08, 17.1) mm, rotated rx 180 ry 0 rz -180 deg; joints [1.365, 66.221, -28.161, 2.214, -38.081, -1.743]
  Call Extruder 0.10099
  MoveL (T15681) to (121.16, 114.41, 17.1) mm, rotated rx 180 ry 0 rz -180 deg; joints [1.365, 66.221, -28.161, 2.214, -38.081, -1.743]
  Call Extruder 0.0177
  MoveL (T15682) to (121.16, 114.99, 17.1) mm, rotated rx 180 ry 0 rz -180 deg; joints [1.365, 66.221, -28.161, 2.214, -38.081, -1.743]
  Call Extruder 0.11352
  MoveL (T15683) to (118.53, 112.36, 17.1) mm, rotated rx 180 ry 0 rz -180 deg; joints [1.319, 71.395, -37.889, 2.389, -33.529, -1.992]
  Call Extruder 0.01252
  MoveL (T15684) to (118.24, 112.65, 17.1) mm, rotated rx 180 ry 0 rz -180 deg; joints [1.319, 71.395, -37.889, 2.389, -33.529, -1.992]
  Call Extruder 0.12605
  MoveL (T15685) to (121.16, 115.56, 17.1) mm, rotated rx 180 ry 0 rz -180 deg; joints [3.282, 71.633, -38.338, 5.963, -33.438, -4.981]
  Call Extruder 0.0177
  MoveL (T15686) to (121.16, 116.14, 17.1) mm, rotated rx 180 ry 0 rz -180 deg; joints [3.282, 71.633, -38.338, 5.963, -33.438, -4.981]
  Call Extruder 0.14418
  MoveL (T15687) to (117.82, 112.81, 17.1) mm, rotated rx 180 ry 0 rz -180 deg; joints [3.398, 66.318, -28.343, 5.511, -38.104, -4.342]
  Set speed (45.0 mm/s)
  Call Extruder -1.6
  MoveL (T15688) to (117.82, 112.81, 17.1) mm, rotated rx 180 ry 0 rz -180 deg; joints [3.398, 66.318, -28.343, 5.511, -38.104, -4.342]
  Set speed (120.0 mm/s)
  MoveL (T15689) to (117.82, 112.81, 17.1) mm, rotated rx 180 ry 0 rz -180 deg; joints [3.398, 66.318, -28.343, 5.511, -38.104, -4.342]
  Call Extruder -0.38
  MoveL (T15690) to (118.58, 113.57, 17.1) mm, rotated rx 180 ry 0 rz -180 deg; joints [1.366, 66.119, -27.969, 2.211, -38.171, -1.739]
  Set speed (45.0 mm/s)
  Call Extruder -0.02
  MoveL (T15691) to (118.58, 113.57, 17.1) mm, rotated rx 180 ry 0 rz -180 deg; joints [1.365, 66.206, -28.132, 2.214, -38.095, -1.742]
  Set speed (150.0 mm/s)
  MoveL (T15692) to (118.58, 113.57, 19.1) mm, rotated rx 180 ry 0 rz -180 deg; joints [1.365, 66.206, -28.132, 2.214, -38.095, -1.742]
  MoveL (T15693) to (121.34, 116.91, 19.1) mm, rotated rx 180 ry 0 rz -180 deg; joints [1.332, 66.014, -27.771, 2.152, -38.263, -1.69]
  MoveL (T15694) to (121.34, 116.91, 17.1) mm, rotated rx 180 ry 0 rz -180 deg; joints [1.332, 66.014, -27.771, 2.152, -38.263, -1.69]
  Set speed (40.0 mm/s)
  Call Extruder 2.0
  MoveL (T15695) to (121.34, 116.91, 17.1) mm, rotated rx 180 ry 0 rz -180 deg; joints [1.332, 66.014, -27.771, 2.152, -38.263, -1.69]
  Call Extruder 0.56525
  MoveL (T15696) to (108.28, 103.84, 17.1) mm, rotated rx 180 ry 0 rz -180 deg; joints [1.332, 66.014, -27.771, 2.152, -38.263, -1.69]
  Call Extruder 0.0177
  MoveL (T15697) to (107.7, 103.84, 17.1) mm, rotated rx 180 ry 0 rz -180 deg; joints [1.332, 66.014, -27.771, 2.152, -38.263, -1.69]
  Call Extruder 0.58235
  MoveL (T15698) to (121.16, 117.3, 17.1) mm, rotated rx 180 ry 0 rz -180 deg; joints [1.332, 66.014, -27.771, 2.152, -38.263, -1.69]
  Call Extruder 0.0177
  MoveL (T15699) to (121.16, 117.88, 17.1) mm, rotated rx 180 ry 0 rz -180 deg; joints [1.332, 66.014, -27.771, 2.152, -38.263, -1.69]
  Call Extruder 0.60738
  MoveL (T15700) to (107.12, 103.84, 17.1) mm, rotated rx 180 ry 0 rz -180 deg; joints [1.332, 66.014, -27.771, 2.152, -38.263, -1.69]
  Call Extruder 0.01156
  MoveL (T15701) to (106.74, 103.84, 17.1) mm, rotated rx 180 ry 0 rz -180 deg; joints [1.323, 66.013, -27.77, 2.137, -38.263, -1.678]
  Call Extruder 0.00434
  MoveL (T15702) to (106.64, 103.94, 17.1) mm, rotated rx 180 ry 0 rz -180 deg; joints [1.276, 71.521, -38.126, 2.317, -33.416, -1.934]
  Call Extruder 0.62807
  MoveL (T15703) to (121.16, 118.46, 17.1) mm, rotated rx 180 ry 0 rz -180 deg; joints [1.276, 71.521, -38.126, 2.317, -33.416, -1.934]
  Call Extruder 0.0177
  MoveL (T15704) to (121.16, 119.03, 17.1) mm, rotated rx 180 ry 0 rz -180 deg; joints [3.322, 71.771, -38.597, 6.054, -33.321, -5.065]
  Call Extruder 0.64059
  MoveL (T15705) to (106.36, 104.23, 17.1) mm, rotated rx 180 ry 0 rz -180 deg; joints [3.322, 71.771, -38.597, 6.054, -33.321, -5.065]
  Call Extruder 0.01252
  MoveL (T15706) to (106.07, 104.52, 17.1) mm, rotated rx 180 ry 0 rz -180 deg; joints [3.322, 71.771, -38.597, 6.054, -33.321, -5.065]
  Call Extruder 0.6531
  MoveL (T15707) to (121.16, 119.61, 17.1) mm, rotated rx 180 ry 0 rz -180 deg; joints [3.322, 71.771, -38.597, 6.054, -33.321, -5.065]
  Call Extruder 0.01604
  MoveL (T15708) to (121.16, 120.14, 17.1) mm, rotated rx 180 ry 0 rz -180 deg; joints [3.322, 71.771, -38.597, 6.054, -33.321, -5.065]
  Call Extruder 0.00167
  MoveL (T15709) to (121.1, 120.14, 17.1) mm, rotated rx 180 ry 0 rz -180 deg; joints [3.445, 66.22, -28.159, 5.576, -38.193, -4.388]
  Call Extruder 0.66326
  MoveL (T15710) to (105.78, 104.81, 17.1) mm, rotated rx 180 ry 0 rz -180 deg; joints [3.445, 66.22, -28.159, 5.576, -38.193, -4.388]
  Call Extruder 0.01252
  MoveL (T15711) to (105.49, 105.1, 17.1) mm, rotated rx 180 ry 0 rz -180 deg; joints [3.445, 66.22, -28.159, 5.576, -38.193, -4.388]
  Call Extruder 0.65064
  MoveL (T15712) to (120.52, 120.14, 17.1) mm, rotated rx 180 ry 0 rz -180 deg; joints [1.339, 66.014, -27.772, 2.162, -38.262, -1.698]
  Call Extruder 0.01772
  MoveL (T15713) to (119.94, 120.14, 17.1) mm, rotated rx 180 ry 0 rz -180 deg; joints [1.339, 66.014, -27.772, 2.162, -38.262, -1.698]
  Call Extruder 0.62639
  MoveL (T15714) to (105.47, 105.66, 17.1) mm, rotated rx 180 ry 0 rz -180 deg; joints [1.339, 66.014, -27.772, 2.162, -38.262, -1.698]
  Call Extruder 0.0177
  MoveL (T15715) to (105.47, 106.24, 17.1) mm, rotated rx 180 ry 0 rz -180 deg; joints [1.326, 66.029, -27.799, 2.142, -38.249, -1.682]
  Call Extruder 0.61188
  MoveL (T15716) to (119.61, 120.38, 17.1) mm, rotated rx 180 ry 0 rz -180 deg; joints [1.326, 66.029, -27.799, 2.142, -38.249, -1.682]
  Call Extruder 0.01252
